		IF rtExecute.Q 
		THEN
			Busy 											:= TRUE;
			Done											:= FALSE;
			Error											:= FALSE;
			ErrorID											:= 0;
			Errortext										:= '';
			CurrState										:= 0;
			linkState										:= 0;
			ReqStateOK										:= FALSE;
			MEMSET(ADR(StateBits),0,SIZEOF(StateBits));
			MEMSET(ADR(CrcError),0,SIZEOF(CrcError));	
			StateText										:= '';
	
			SetSlaveSTATE(bExecute := FALSE, sNetId:= EcMasterAmsNetId,nSlaveAddr:= SlaveAddr);
			GetSlaveSTATE(bExecute := FALSE,sNetId:= EcMasterAmsNetId,nSlaveAddr:= SlaveAddr);
			GetSlaveCrcErrorEx(bExecute := FALSE,sNetId:= EcMasterAmsNetId,nSlaveAddr:= SlaveAddr);

			IF(ReqState <> CurrState
				OR ReqState <> MemReqState)
				AND ReqState <> 0
			THEN
				SetSlaveState(bExecute:= TRUE,reqState:= ReqState);
				MemReqState 								:= ReqState;
				state 										:= 10;

			ELSE
				(* Start Reading State *)
				GetSlaveState(bExecute	:= TRUE);
				state 										:= 1;
			END_IF

		ELSIF NOT Execute 
		THEN
			Done 											:= FALSE;
			Error											:= FALSE;
			ErrorID											:= 0;
			ErrorText										:= '';
		END_IF

	(* Read Slave State **************************************)
	1:
		(* Work block *)
		GetSlaveState();

		IF NOT GetSlaveState.bBusy
		THEN
			IF GetSlaveState.bError THEN
				Busy										:= FALSE;
				Error										:= TRUE;
				ErrorId										:= GetSlaveState.nErrId;
				ErrorText									:= CONCAT('FB_EcGetSlaveSTATE Id: ',UDINT_TO_STRING(ErrorId));
				state 										:= 0;
			ELSE       
				ReqStateOK 									:= (ReqState = CurrState OR ReqState = 0);         					
				CurrState 									:= GetSlaveState.state.deviceState;
				linkState 									:= GetSlaveState.State.linkState;
				StateText 									:= F_ConvStateToString(GetSlaveState.State.deviceState);
			 	StateBits							 		:= F_ConvSlaveStateToBitsEx(GetSlaveState.state);
				state										:= state + 1;
			END_IF
			GetSlaveSTATE(bExecute := FALSE);
		ELSE
			;
		END_IF

	(* Read Slave CRC Error Counter  **************************************)		
	2: 
		(* Work block *)
		GetSlaveCrcErrorEx();

		IF NOT GetSlaveCrcErrorEx.bBusy
		THEN
			IF GetSlaveCrcErrorEx.bError THEN
				Busy										:= FALSE;
				Error										:= TRUE;
				ErrorId										:= GetSlaveCrcErrorEx.nErrId;
				ErrorText									:= CONCAT('FB_EcGetSlaveCrcErrorEx Id: ',UDINT_TO_STRING(ErrorId));
				state 										:= 0;
			ELSE       
				CrcError									:= 	GetSlaveCrcErrorEx.crcError;
				Done 										:= TRUE;
				Busy 										:= FALSE;
				state										:= 0;
			END_IF
			GetSlaveCrcErrorEx(bExecute := FALSE);
		ELSE
			;
		END_IF

	(* Set state  *****************************************)
	10:	
		SetSlaveState();  
		IF NOT SetSlaveState.bBusy
		THEN
			IF SetSlaveState.bError 
			THEN             	
				Busy										:= FALSE;
				Error										:= TRUE;
				ErrorId										:= SetSlaveState.nErrId;
				ErrorText									:= CONCAT('FB_EcSetSlaveSTATE Id: ',UDINT_TO_STRING(ErrorId));
				state 										:= 0;
			ELSIF SetSlaveState.CurrState.deviceState = MemReqState 
			THEN
				ReqStateOK									:= TRUE;
				Busy 										:= FALSE;
				Done 										:= TRUE;	
				state 										:= 0;
			ELSE                    				
				Busy										:= FALSE;		
				Error										:= TRUE;
				ErrorId										:= E_AdsErr.DEVICE_ABORTED;
				ErrorText									:= 'SetSlaveState DEVICESTATE <> ReqState';
				state	 									:= 0;
			END_IF         					
			CurrState 										:= SetSlaveState.currState.deviceState;
			linkState 										:= SetSlaveState.currState.linkState;
			StateText 										:= F_ConvStateToString(SetSlaveState.currState.deviceState);
			StateBits							 			:= F_ConvSlaveStateToBitsEx(SetSlaveState.currState);
			SetSlaveState(bExecute := FALSE);              						
		END_IF                      						
	END_CASE


(*********************************************************************)

END_FUNCTION_BLOCK

// ---- POUs/FileHandling/Basic/FileHandling.TcPOU
{attribute 'no_check'}
//Wrapper for all file fucntions provided by lib Tc2_TcSystem.Lib, see Beckhoff information system for detailed information of each function. 
FUNCTION_BLOCK FileHandling EXTENDS FbBase
VAR_OUTPUT CONSTANT
	FNC_OPEN												:	INT := 0; //With this function a new file can be created, or a closed existing file can be re-opened for further processing
	FNC_READ												:	INT := 1; //With this function  the contents of an already opened file can be read. The file must have been already opened for read access
	FNC_WRITE												:	INT := 2; //Data can be written into a file with this function if it is opened in write mode
	FNC_PUTS												:	INT := 3; //The function writes strings to the file if it is opened in write mode
	FNC_GETS												:	INT := 4; //The function reads zero terminated strings from a file and moves the file pointer to the next line.(if pBuffer is <> 0, the read line will copied to the buffer as well)
	FNC_CLOSE												:	INT := 5; //With this function the file can be closed, and thereby placed into a defined state for further processing by other programs
	FNC_DELETE												:	INT := 6; //With this function the existing file can be deleted
	FNC_RENAME												:	INT := 7; //With this function the existing file can be renamed.
	FNC_REMOVEDIR											:	INT := 8; //This function removes a directory from the data medium. A directory containing data can not be removed!
	FNC_CREATEDIR											:	INT := 9; //This function creates new directories on the data medium.
	FNC_SEEK												:	INT := 10;//With this function the file pointer of an opened file can be set to a definable position
	FNC_TELL												:	INT := 11;//The function gets the current position of the file pointer. The position is expressed as an offset relative to the beginning of the stream.
	FNC_EOF													:	INT := 12;//The function tests for the end-of-file.
	FNC_LOAD												:	INT := 13;//The file is opened implicitly in binary mode, the contents are read out and the file is then closed again.
END_VAR             										                 										
VAR_INPUT           										
	Fnc														:	INT (FNC_OPEN..FNC_LOAD) := FNC_OPEN; //Parameter for requested function
	AMSNetId												:	T_AmsNetId := ''; //Ams Net Id 
	Timeout													:	TIME := DEFAULT_ADS_TIMEOUT; //Ads timeout 
	Mode													:	DWORD := FOPEN_MODEAPPEND OR FOPEN_MODEPLUS OR FOPEN_MODETEXT; 
																			(* 	FOPEN_MODEREAD "r": Opens for reading. If the file does not exist or cannot be found, the call fails.
																				FOPEN_MODEWRITE  "w": Opens an empty file for writing. If the given file exists, its contents are destroyed.
																				FOPEN_MODEAPPEND  "a": Opens for writing at the end of the file (appending) without removing the EOF marker before writing new data to the file; creates the file first if it doesn’t exist.
																				FOPEN_MODEREAD OR FOPEN_MODEPLUS  "r+": Opens for reading and writing. The file must exist.
																				FOPEN_MODEWRITE OR FOPEN_MODEPLUS  "w+": Opens an empty file for both reading and writing. If the given file exists, its contents are destroyed.
																				FOPEN_MODEAPPEND OR FOPEN_MODEPLUS  "a+": 	Opens for reading and appending; the appending operation includes the removal of the EOF marker before new data is written to the file and the EOF marker is restored after writing is complete; creates the file first if it doesn’t exist.
																															When a file is opened with the "a" or "a+" access type, all write operations occur at the end of the file. The file pointer can be repositioned using FB_FileSeek, but is always moved back to the end of the file before any write operation is carried out. Thus, existing data cannot be overwritten. 																				                                    								
																				FOPEN_MODEBINARY  "b": Open in binary (untranslated) mode.
																				FOPEN_MODETEXT  "t": Open in text (translated) mode. *)
	Path													:	T_MaxString; // \\PC-Name\Folder\ 
	FileName												:	T_MaxString := ''; // NewFile.xyz 
	OldFileName												:	T_MaxString := ''; // File.xyz 
	pBuffer													:	PVOID; //pointer to data section 
	Length													: 	UDINT; // sizeof data section for read and write. Note to use "LEN" while writing-command, beacause otherwise the whole datasection and not only the string will be written 
	SeekOrigin												: 	E_SeekOrigin := SEEK_SET; //Seek function parameter - Contains the relative position for the move.
	SeekPos													:	DINT; //Seek function parameter - Contains the desired (new) target position of the file pointer.
END_VAR
VAR_OUTPUT
	EOF														:	BOOL;	//This output is switched to TRUE if the end of file is reached.
	WorkedLen												:	UDINT;	//Contains the number of bytes currently read or written
	hFile													:	UINT;	//File handle of currently opened file
	ActSeekPos												:	DINT;	//Act file pointer position of filled by Tell function
	Line   													: T_MaxString; //Read line of file - filled by function Gets

END_VAR
VAR
(* internal used variables ************************************************************)
	MemErrorText											:	STRING(50);
	MemFnc													:	INT := -1;
	
(* trigger ******************************************************************************)

(* function-block instances ************************************************************)
	File_Open												:	FB_FileOpen;
	File_Close												: 	FB_FileClose;
	File_Read 												: 	FB_FileRead;
	File_Write												:	FB_FileWrite;
	File_Delete												:	FB_FileDelete;
	File_Rename												:	FB_FileRename;
	File_Puts												:	FB_FilePuts;
	File_Gets												:	FB_FileGets;
	File_CreateDir											:	FB_CreateDir;
	File_RemoveDir											:	FB_RemoveDir;
	File_Tell												:	FB_FileTell ;
	File_Seek												:	FB_FileSeek ;
	File_EoF												:	FB_EOF;
	File_Load												:	FB_FileLoad;
END_VAR

	(* FileHandling												V2.0	*)
	(********************************************************************)

(* Sequence **********************************************************************)
	rtExecute(CLK := Execute);
	IF rtExecute.Q
		AND MemFnc < 0
	THEN
		Busy												:= TRUE;
		Done												:= FALSE;
		Error												:= FALSE;
		ErrorId												:= 0;
		CASE fnc OF                     					
		FNC_OPEN:		MemFnc 								:= fnc;
		FNC_READ:		MemFnc 								:= fnc;
		FNC_WRITE:		MemFnc 								:= fnc;
		FNC_PUTS:		MemFnc 								:= fnc;
		FNC_GETS:		MemFnc 								:= fnc;
		FNC_CLOSE:		MemFnc 								:= fnc;
		FNC_DELETE:		MemFnc 								:= fnc;
		FNC_RENAME:		MemFnc 								:= fnc;
		FNC_REMOVEDIR: 	MemFnc 								:= fnc;
		FNC_CREATEDIR: 	MemFnc 								:= fnc;
		FNC_SEEK:		MemFnc 								:= fnc;
		FNC_TELL:		MemFnc 								:= fnc;
		FNC_EOF:		MemFnc 								:= fnc;
		FNC_LOAD:		MemFnc 								:= fnc;
		ELSE                            					
			ErrorId											:= E_AdsErr.DEVICE_INVALIDPARM;
			Error											:= TRUE;
			Done											:= FALSE;
			Busy											:= FALSE;
		END_CASE
	END_IF

	CASE MemFnc OF
		FNC_OPEN:		Open(Execute := Execute);
		FNC_READ:		Read(Execute := Execute);
		FNC_WRITE:		Write(Execute := Execute);
		FNC_PUTS:		Puts(Execute := Execute);
		FNC_GETS:		Gets(Execute := Execute);
		FNC_CLOSE:		Close(Execute := Execute);
		FNC_DELETE:		Delete(Execute := Execute);
		FNC_RENAME:		Rename(Execute := Execute);
		FNC_REMOVEDIR: 	RemoveDir(Execute := Execute);
		FNC_CREATEDIR: 	CreateDir(Execute := Execute);
		FNC_SEEK:		Seek(Execute := Execute);
		FNC_TELL:		Tell(Execute := Execute);
		FNC_EOF:		IsEof(Execute := Execute);
		FNC_LOAD:		Load(Execute := Execute);
	
	-1:
		IF NOT Execute
		THEN
			Busy											:= FALSE;
			Done											:= FALSE;
			Error											:= FALSE;
			ErrorID											:= 0;
		END_IF
	END_CASE
(*************************************************************************)

METHOD PUBLIC close : Bool //Return value = TRUE if busy
VAR_INPUT
	Execute		:	BOOL	:= FALSE;
END_VAR
	IF Execute
	THEN
		Error												:=	FALSE;
		ErrorId												:= 0;
		File_Close.bExecute 								:= TRUE;
	ELSIF NOT File_Close.bBusy      						
	THEN                            						
		Error												:=	FALSE;
		ErrorId												:= 0;
		File_Close.bExecute 								:= FALSE;
	END_IF                          						
                                    	
	MemFnc 													:= FNC_CLOSE;
	THIS^.Execute											:= Execute;

	File_Close(
		sNetId		:= AMSNetId,
		hFile		:= hFile,
		bExecute	:= ,
		tTimeout	:= Timeout,
		bBusy		=> Busy,
		bError		=> ,
		nErrId		=> );

	IF NOT File_Close.bBusy
		AND NOT File_Close.bError
		AND File_Close.bExecute
	THEN
		Done												:= TRUE;
		hFile 												:= 0;
	ELSE                            						
		Done												:= FALSE;
	END_IF

	IF NOT Busy
	THEN
		IF File_Close.bExecute
		THEN
			Error											:=	File_Close.bError;
			ErrorId											:= File_Close.nErrId;
		END_IF
		IF NOT Execute
		THEN
			MemFnc											:=  -1;
			File_Close(bExecute 							:= FALSE);
		END_IF
	END_IF

	(* Fehler speichern *)
	IF Error
	THEN
		MemErrorText										:= CONCAT('File_Close ErrorID: ', UDINT_TO_STRING(ErrorID));
	END_IF
	
	Close													:= Busy;
END_METHOD

METHOD PUBLIC createDir : BOOL //Return value = TRUE if busy
//required parameter
//Path
VAR_INPUT
	Execute													:	BOOL;
END_VAR
	IF Execute
	THEN
		Error												:=	FALSE;
		ErrorId												:= 0;
		File_CreateDir.bExecute 							:= TRUE;
	ELSIF NOT File_CreateDir.bBusy      					
	THEN                                					
		Error												:=	FALSE;
		ErrorId												:= 0;
		File_CreateDir.bExecute								:= FALSE;
	END_IF                              					
                                        	
	MemFnc 													:= FNC_CREATEDIR;
	THIS^.Execute											:= Execute;

	File_CreateDir(
		sNetId		:= AMSNetId,
		sPathName	:= Path,
		ePath		:= ,
		bExecute	:= ,
		tTimeout	:= Timeout,
		bBusy		=> Busy,
		bError		=> ,
		nErrId		=> );

	Done													:= NOT File_CreateDir.bBusy
																AND NOT File_CreateDir.bError
																AND File_CreateDir.bExecute;
	IF NOT Busy
	THEN
		IF File_CreateDir.bExecute
		THEN
			Error											:=	File_CreateDir.bError;
			ErrorId											:= File_CreateDir.nErrId;
		END_IF
		IF NOT Execute
		THEN
			MemFnc											:=  -1;
			File_CreateDir(bExecute := FALSE);
		END_IF
	END_IF


	IF Error
	THEN
		MemErrorText										:= CONCAT('File_CreateDir ErrorID: ', UDINT_TO_STRING(ErrorID));
	END_IF
	
	CreateDir												:= Busy;
END_METHOD

METHOD PUBLIC delete : BOOL //Return value = TRUE if busy
//required parameter
//Path
//FileName
VAR_INPUT
	Execute			:	bool;
END_VAR
	IF Execute
	THEN
		Error												:=	FALSE;
		ErrorId												:= 0;
		File_Delete.bExecute 								:= TRUE;
	ELSIF NOT File_Delete.bBusy         					
	THEN                                					
		Error												:=	FALSE;
		ErrorId												:= 0;
		File_Delete.bExecute 								:= FALSE;
	END_IF                              					
                                        	
	MemFnc 													:= FNC_DELETE;
	THIS^.Execute											:= Execute;

	File_Delete(
		sNetId		:= AMSNetId,
		sPathName	:= CONCAT(Path,FileName),
		ePath		:= ,
		bExecute	:= ,
		tTimeout	:= Timeout,
		bBusy		=> Busy,
		bError		=> ,
		nErrId		=> );

	Done													:= 	NOT File_Delete.bBusy
																AND NOT File_Delete.bError
																AND File_Delete.bExecute;
	IF NOT Busy
	THEN
		IF File_Delete.bExecute
		THEN
			Error											:=	File_Delete.bError;
			ErrorId											:= File_Delete.nErrId;
		END_IF
		IF NOT Execute
		THEN
			MemFnc											:= -1;
			File_Delete(bExecute := FALSE);
		END_IF
	END_IF


	IF Error
	THEN
		MemErrorText										:= CONCAT('File_Delete ErrorID: ', UDINT_TO_STRING(ErrorID));
	End_if
	
	Delete													:= Busy;
END_METHOD

METHOD PUBLIC gets : BOOL //Return value = TRUE if busy
//required parameter
//Path
//Filename
//Mode
//pBuffer
VAR_INPUT
	Execute			:	BOOL;
END_VAR
IF pBuffer = 0 THEN
	Busy													:= NOT Error;
	Error													:= TRUE;
	ErrorId													:= E_AdsErr.DEVICE_INVALIDPARM;
	Done													:= FALSE;
	MemFnc													:= -1 ;
	RETURN;                             					
END_IF                                  					
                                        					
	MemFnc 													:= FNC_GETS;
	THIS^.Execute											:= Execute;
                                        					
	CASE State OF                       	
	0:                                  	
		IF Execute                      	
		THEN                            	
			Done											:= FALSE;
			Error											:= FALSE;
			ErrorId 										:= 0;
			
			File_Open(bExecute := FALSE);
			File_Gets(bExecute := FALSE);
			File_Close(bExecute := FALSE);
			
			EOF												:= FALSE;
			WorkedLen										:= 0;
			
			IF hFile = 0
			THEN
				File_Open(
					sNetId		:= AMSNetId,
					sPathName	:= CONCAT(Path,FileName),
					nMode		:= Mode ,
					ePath		:= (* Default *),
					bExecute	:= TRUE,
					tTimeout	:= Timeout,
					bBusy		=> ,
					bError		=> ,
					nErrId		=> ,
					hFile		=> );

				State 										:= 10;
			ELSE                							
				State 										:= 10;
			END_IF
		ELSE
			Done											:= FALSE;
			Error											:= FALSE;
			ErrorId 										:= 0;
		END_IF

	10:
		File_Open();

		IF NOT File_Open.bBusy
		THEN
			IF File_Open.bError
			THEN
				State 										:= 99;
			ELSE
				IF File_Open.bExecute THEN hFile := File_Open.hFile; END_IF
				File_Gets(
					sNetId		:= AMSNetId,
					hFile		:= hFile,
					bExecute	:= TRUE,
					tTimeout	:= Timeout,
					sLine		=> ,
					bEOF		=> ,
					bBusy		=> ,
					bError		=> ,
					nErrId		=> );

				State 										:= 20;
			END_IF
		END_IF

	20:
		File_Gets(bEOF		=> EOF);
		IF NOT File_Gets.bBusy
		THEN
			IF NOT File_Gets.bError
			THEN
				IF pBuffer <> 0 AND Length <> 0
				THEN
					 MEMCPY(pBuffer , ADR(File_Gets.sLine), MIN(TO_UDINT(Length), SIZEOF(File_Gets.sLine)));
				END_IF
				Line										:= File_Gets.sLine;
			END_IF
			IF File_Open.bExecute
			THEN
				File_Close(
					sNetId	:= AMSNetId,
					hFile	:= hFile,
					bExecute:= TRUE,
					tTimeout:= Timeout,
					bBusy	=> ,
					bError	=> ,
					nErrId	=> );
				State										:= 30;
			ELSE
				State										:= 99;
			END_IF

		END_IF

	30:
		File_Close();
		IF NOT File_Close.bBusy
		THEN
			hFile											:= 0;
			State											:= 99;
		END_IF

	99:
		IF NOT Execute
		THEN
			Memfnc											:= -1;
			state 											:= 0;
		END_IF
	END_CASE

	Done													:= state = 99
																AND NOT File_Gets.bError
																AND NOT File_Close.bError
																AND NOT File_Open.bError;
                                        					
	Error													:= state = 99
																AND(
																File_Gets.bError
																OR File_Close.bError
																OR File_Open.bError);
                                        					
	Busy													:= state <> 0
																AND NOT Done
																AND NOT Error;

	IF Error
	THEN
		IF File_Close.bError 	THEN 	ErrorId :=  File_Close.nErrId; 	END_IF
		IF File_Gets.bError 	THEN 	ErrorId :=  File_Gets.nErrId; 	END_IF
		IF File_Open.bError 	THEN	ErrorId :=  File_Open.nErrId; 	END_IF
	ELSE
		ErrorId 											:= 0;
	END_IF                              					
                                        					
	IF NOT Execute                      					
		AND state = 99                  					
	THEN                                					
			MemFnc											:= -1;
		state 												:= 0;
	END_IF                              	
                                        	
	IF Error                            	
	THEN                                	
		MemErrorText										:= CONCAT('File_Gets ErrorID: ', UDINT_TO_STRING(ErrorID));
	END_IF                              					
                                        					
	Gets													:= Busy;
END_METHOD

METHOD PUBLIC isEoF : BOOL //Return value = TRUE if busy
VAR_INPUT
	Execute													:	BOOL;
END_VAR
	IF Execute
	THEN
		Error												:=	FALSE;
		ErrorId												:= 0;
		File_EoF.bExecute 									:= TRUE;
	ELSIF NOT File_EoF.bBusy           					
	THEN                                					
		Error												:=	FALSE;
		ErrorId												:= 0;
		File_EoF.bExecute 									:= FALSE;
	END_IF                              							
	                                    	
	MemFnc 													:= FNC_EOF;
	THIS^.Execute											:= Execute;
                                        	
	File_EoF(
		sNetId		:= AMSNetId,
		hFile		:= hFile ,
		tTimeout	:= Timeout,
		bBusy		=> Busy,
		bError		=> ,
		nErrId		=> ,
		bEoF		=> EoF);

	Done													:= NOT File_EoF.bBusy
																AND NOT File_EoF.bError
																AND File_EoF.bExecute;
	IF NOT Busy                         					
	THEN                        					
		IF File_EoF.bExecute           					
		THEN                            	
			Error											:=	File_EoF.bError;
			ErrorId											:= File_EoF.nErrId;
		END_IF
		IF NOT Execute
		THEN
			MemFnc											:= 1;
			File_EoF(bExecute := FALSE);
		END_IF
	END_IF


	IF Error
	THEN
		MemErrorText										:= CONCAT('File_EoF ErrorID: ', UDINT_TO_STRING(ErrorID));
	END_IF
	
	IsEoF													:= Busy;
END_METHOD

METHOD PUBLIC load : BOOL //Result = Busy
//required parameter
//Path
//FileName
VAR_INPUT
	Execute				:	BOOL; 
END_VAR
IF Execute
THEN
	Error													:= FALSE;
	ErrorId													:= 0;
	File_Load.bExecute 										:= TRUE;
ELSIF NOT File_Load.bBusy           						
THEN                                						
	Error													:=	FALSE;
	ErrorId													:= 0;
	File_Load.bExecute 										:= FALSE;
END_IF	

MemFnc 														:= FNC_LOAD;
THIS^.Execute												:= Execute;

(* Work File Load *)
File_Load(
	sNetId		:= AMSNetId, 
	sPathName	:= CONCAT(Path,FileName), 
	pReadBuff	:= pBuffer, 
	cbReadLen	:= Length, 
	bExecute	:= , 
	tTimeout	:= Timeout, 
	bBusy		=> Busy, 
	bError		=> , 
	nErrId		=> , 
	cbRead		=> WorkedLen);
Done														:= NOT File_Load.bBusy
																AND NOT File_Load.bError
																AND File_Load.bExecute;
IF NOT Busy
THEN
	IF File_Load.bExecute
	THEN
		Error												:= File_Load.bError;
		ErrorId												:= File_Load.nErrId;
	END_IF
	IF NOT Execute
	THEN
		MemFnc												:= -1;
		File_Load(bExecute := FALSE);
	END_IF
END_IF

IF Error
THEN
	MemErrorText											:= CONCAT('File_Load ErrorID: ', UDINT_TO_STRING(ErrorID));
END_IF                              						
                                    	
load														:= Busy;
END_METHOD

METHOD PUBLIC open : BOOL //Return value = TRUE if busy
//required parameter
//Path
//FileName
//Mode
VAR_INPUT
	Execute				:	BOOL; 
END_VAR
IF Execute
THEN
	Error													:= FALSE;
	ErrorId													:= 0;
	File_Open.bExecute 										:= TRUE;
ELSIF NOT File_Open.bBusy           						
THEN                                						
	Error													:=	FALSE;
	ErrorId													:= 0;
	File_Open.bExecute 										:= FALSE;
END_IF	

MemFnc 														:= FNC_OPEN;
THIS^.Execute												:= Execute;

(* Work File Open *)
File_Open(
	sNetId		:= AMSNetId,
	sPathName	:= CONCAT(Path,FileName),
	nMode		:= Mode ,
	ePath		:= (* Default *),
	bExecute	:= ,
	tTimeout	:= Timeout,
	bBusy		=> Busy,
	bError		=> ,
	nErrId		=> ,
	hFile		=> hFile);

Done														:= NOT File_Open.bBusy
																AND NOT File_Open.bError
																AND File_Open.bExecute;
IF NOT Busy
THEN
	IF File_Open.bExecute
	THEN
		Error												:=	File_Open.bError;
		ErrorId												:= File_Open.nErrId;
	END_IF
	IF NOT Execute
	THEN
		MemFnc												:= -1;
		File_Open(bExecute := FALSE);
	END_IF
END_IF

IF Error
THEN
	MemErrorText											:= CONCAT('File_Open ErrorID: ', UDINT_TO_STRING(ErrorID));
END_IF                              						
                                    	
Open														:= Busy;
END_METHOD

METHOD PUBLIC puts : BOOL //Return value = TRUE if busy
//required parameter
//Path
//FileName
//Mode
//pBuffer
//Lenght
VAR_INPUT
	Execute				:	BOOL;
END_VAR
IF pBuffer = 0 THEN
	Busy													:= NOT Error;
	Error													:= TRUE;
	ErrorId													:= E_AdsErr.DEVICE_INVALIDPARM;
	Done													:= FALSE;
	MemFnc													:= -1 ;
	RETURN;
END_IF

	MemFnc 													:= FNC_PUTS;
	THIS^.Execute											:= Execute;

	CASE State OF
	0:
		IF Execute
		THEN
			Done											:= FALSE;
			Error											:= FALSE;
			ErrorId 										:= 0;
			
			File_Open(bExecute := FALSE);
			File_Puts(bExecute := FALSE);
			File_Close(bExecute := FALSE);
			
			EOF												:= FALSE;
			WorkedLen										:= 0;
			
			IF hFile = 0
			THEN
				File_Open(
					sNetId		:= AMSNetId,
					sPathName	:= CONCAT(Path,FileName),
					nMode		:= Mode ,
					ePath		:= (* Default *),
					bExecute	:= TRUE,
					tTimeout	:= Timeout,
					bBusy		=> ,
					bError		=> ,
					nErrId		=> ,
					hFile		=> );

				State 										:= 10;
			ELSE                							
				State 										:= 10;
			END_IF              							
		ELSE                    							
			Done											:= FALSE;
			Error											:= FALSE;
			ErrorId 										:= 0;
		END_IF

	10:
		File_Open();

		IF NOT File_Open.bBusy
		THEN
			IF File_Open.bError
			THEN
				State 										:= 99;
			ELSE
				IF File_Open.bExecute THEN hFile := File_Open.hFile; END_IF
				MEMCPY(ADR(File_Puts.sLine),  pBuffer, MIN(TO_UDINT(Length), SIZEOF(File_Puts.sLine)));
				File_Puts(
					sNetId		:= AMSNetId,
					hFile		:= hFile,
					sLine		:= (* siehe oben *),
					bExecute	:= TRUE,
					tTimeout	:= Timeout,
					bBusy		=> ,
					bError		=> ,
					nErrId		=> );

				State 										:= 20;
			END_IF
		END_IF

	20:
		MEMCPY(ADR(File_Puts.sLine),  pBuffer, MIN(TO_UDINT(Length), SIZEOF(File_Puts.sLine)));
		File_Puts();

		IF NOT File_Puts.bBusy
		THEN
			IF File_Open.bExecute
			THEN
				File_Close(
					sNetId	:= AMSNetId,
					hFile	:= hFile,
					bExecute:= TRUE,
					tTimeout:= Timeout,
					bBusy	=> ,
					bError	=> ,
					nErrId	=> );
				State										:= 30;
			ELSE
				State										:= 99;
			END_IF

		END_IF

	30:
		File_Close();
		IF NOT File_Close.bBusy
		THEN
			hFile						:= 0;
			State						:= 99;
		END_IF

	99:
		IF NOT Execute
		THEN
			Memfnc					:= -1;
			state 					:= 0;
		END_IF
	END_CASE

	Done							:= state = 99
										AND NOT File_Puts.bError
										AND NOT File_Close.bError
										AND NOT File_Open.bError;

	Error							:= state = 99
										AND(
										File_Puts.bError
										OR File_Close.bError
										OR File_Open.bError);

	Busy							:= state <> 0
										AND NOT Done
										AND NOT Error;

	IF Error
	THEN
		IF File_Close.bError 	THEN	ErrorId :=  File_Close.nErrId; 	END_IF
		IF File_Puts.bError 	THEN 	ErrorId :=  File_Puts.nErrId; 	END_IF
		IF File_Open.bError 	THEN 	ErrorId :=  File_Open.nErrId;	END_IF
	ELSE
		ErrorId 					:= 0;
	END_IF

	IF NOT Execute
		AND state = 99
	THEN
		MemFnc						:= -1;
		state 						:= 0;
	END_IF

	IF Error
	THEN
		MemErrorText				:= CONCAT('File_Puts ErrorID: ', UDINT_TO_STRING(ErrorID));
	END_IF
	
	Puts							:= Busy;
END_METHOD

METHOD PUBLIC read : BOOL //Return value = TRUE if busy
//required parameter
//Path
//FileName
//Mode
//pBuffer
//Lenght
VAR_INPUT
	Execute			:	BOOL;
END_VAR
IF pBuffer = 0 THEN
	Busy													:= NOT Error;
	Error													:= TRUE;
	ErrorId													:= E_AdsErr.DEVICE_INVALIDPARM;
	Done													:= FALSE;
	MemFnc													:= -1 ;
	RETURN;                             					
END_IF                                  					
                                        	
	MemFnc 													:= FNC_READ;
	THIS^.Execute											:= Execute;

	CASE State OF
	0:
		IF Execute
		THEN
			Done											:= FALSE;
			Error											:= FALSE;
			ErrorId 										:= 0;
			
			File_Open(bExecute := FALSE);
			File_Read(bExecute := FALSE);
			File_Close(bExecute := FALSE);
			
			EOF												:= FALSE;
			WorkedLen										:= 0;
			
			IF hFile = 0
			THEN
				File_Open(
					sNetId		:= AMSNetId,
					sPathName	:= CONCAT(Path,FileName),
					nMode		:= Mode ,
					ePath		:= (* Default *),
					bExecute	:= TRUE,
					tTimeout	:= Timeout,
					bBusy		=> ,
					bError		=> ,
					nErrId		=> ,
					hFile		=> );

				State 										:= 10;
			ELSE                    						
				State 										:= 10;
			END_IF                  						
		ELSE                        						
			Done											:= FALSE;
			Error											:= FALSE;
			ErrorId 										:= 0;
		END_IF

	10:
		File_Open();
		IF NOT File_Open.bBusy
		THEN
			IF File_Open.bError
			THEN
				State 										:= 99;
			ELSE
				IF File_Open.bExecute THEN hFile := File_Open.hFile; END_IF
				File_Read(
					sNetId		:= AmsNetId,
					hFile		:= hFile,
					pReadBuff	:= pBuffer,
					cbReadLen	:= Length,
					bExecute	:= TRUE,
					tTimeout	:= Timeout,
					bBusy		=> ,
					bError		=> ,
					nErrId		=> ,
					cbRead		=> ,
					bEOF		=> );

				State 										:= 20;
			END_IF
		END_IF

	20:
		File_Read(
			pReadBuff	:= pBuffer,
			cbReadLen	:= Length,
			bExecute	:= TRUE,
			cbRead		=> WorkedLen,
			bEOF		=> EOF);

		IF NOT File_Read.bBusy
		THEN
			IF File_Open.bExecute
			THEN
				File_Close(
					sNetId	:= AMSNetId,
					hFile	:= hFile,
					bExecute:= TRUE,
					tTimeout:= Timeout,
					bBusy	=> ,
					bError	=> ,
					nErrId	=> );
				State										:= 30;
			ELSE                        						
				State										:= 99;
			END_IF                      						
                                        						
		END_IF                          						
                                        						
	30:                                 						
		File_Close();                   						
		IF NOT File_Close.bBusy         						
		THEN                            						
			hFile											:= 0;
			State											:= 99;
		END_IF                          						
                                        						
	99:                                 						
		IF NOT Execute                  						
		THEN                            				
			Memfnc											:= -1;
			state 											:= 0;
		END_IF                          	
	END_CASE                            	
                                        	
	Done													:= state = 99
																AND NOT File_Read.bError
																AND NOT File_Close.bError
																AND NOT File_Open.bError;
	                                    						
	Error													:= state = 99
																AND(
																File_Read.bError
																OR File_Close.bError
																OR File_Open.bError);
	                                    						
	Busy													:= state <> 0
																AND NOT Done
																AND NOT Error;

	IF Error
	THEN
		IF File_Close.bError	THEN 	ErrorId :=  File_Close.nErrId;	END_IF
		IF File_Read.bError 	THEN	ErrorId :=  File_Read.nErrId; 	END_IF
		IF File_Open.bError		THEN	ErrorId :=  File_Open.nErrId; 	END_IF
	ELSE
		ErrorId 											:= 0;
	END_IF                              						
                                        						
	IF NOT Execute                      						
		AND state = 99                  						
	THEN                                						
		MemFnc												:=  -1;
		state 												:= 0;
	END_IF                              	
                                        	
	IF Error                            	
	THEN                                	
		MemErrorText										:= CONCAT('File_Read ErrorID: ', UDINT_TO_STRING(ErrorID));
	END_IF                              						
	                                    						
	Read													:= Busy;
END_METHOD

METHOD PUBLIC removeDir : BOOL //Return value = TRUE if busy
//required parameter
//Path
VAR_INPUT
	Execute				:	BOOL;
END_VAR
	IF Execute
	THEN
		Error												:= FALSE;
		ErrorId												:= 0;
		File_RemoveDir.bExecute 							:= TRUE;
	ELSIF NOT File_RemoveDir.bBusy      					
	THEN                                					
		Error												:=	FALSE;
		ErrorId												:= 0;
		File_RemoveDir.bExecute 							:= FALSE;
	END_IF                              					
                                        	
	MemFnc 													:= FNC_REMOVEDIR;
	THIS^.Execute											:= Execute;

	File_RemoveDir(
		sNetId		:= AMSNetId,
		sPathName	:= Path,
		ePath		:= ,
		bExecute	:= ,
		tTimeout	:= Timeout,
		bBusy		=> Busy,
		bError		=> ,
		nErrId		=> );

	Done													:= NOT File_RemoveDir.bBusy
																AND NOT File_RemoveDir.bError
																AND File_RemoveDir.bExecute;
	IF NOT Busy                         					
	THEN                                					
		IF File_RemoveDir.bExecute      					
		THEN                            					
			Error											:=	File_RemoveDir.bError;
			ErrorId											:= File_RemoveDir.nErrId;
		END_IF                          	
		IF NOT Execute                  	
		THEN                            	
			MemFnc											:=  -1;
			File_RemoveDir(bExecute := FALSE);
		END_IF
	END_IF


	IF Error
	THEN
		MemErrorText										:= CONCAT('File_RemoveDir ErrorID: ', UDINT_TO_STRING(ErrorID));
	END_IF                              					
	                                    	
	RemoveDir												:= Busy;
END_METHOD

METHOD PUBLIC rename : BOOL //Return value = TRUE if busy
//required parameter
//Path
//OldFileName
//FileName
VAR_INPUT
	Execute			:	BOOL;
END_VAR
	IF Execute
	THEN
		Error												:=	FALSE;
		ErrorId												:= 0;
		File_Rename.bExecute 								:= TRUE;
	ELSIF NOT File_Rename.bBusy         					
	THEN                                					
		Error												:=	FALSE;
		ErrorId												:= 0;
		File_Rename.bExecute 								:= FALSE;
	END_IF                              					
                                        	
	MemFnc 													:= FNC_RENAME;
	THIS^.Execute											:= Execute;

	File_Rename(
		sNetId		:= AMSNetId,
		sOldName	:= CONCAT(Path,OldFileName),
		sNewName	:= CONCAT(Path,FileName),
		ePath		:= ,
		bExecute	:=	,
		tTimeout	:=	Timeout,
		bBusy		=> Busy,
		bError		=> ,
		nErrId		=> );

	Done													:= NOT File_Rename.bBusy
																AND NOT File_Rename.bError
																AND File_Rename.bExecute;
	IF NOT Busy                         					
	THEN                                					
		IF File_Rename.bExecute         					
		THEN                            	
			Error											:=	File_Rename.bError;
			ErrorId											:= File_Rename.nErrId;
		END_IF
		IF NOT Execute
		THEN
			MemFnc											:= -1;
			File_Rename(bExecute := FALSE);
		END_IF
	END_IF


	IF Error
	THEN
		MemErrorText										:= CONCAT('File_Rename ErrorID: ', UDINT_TO_STRING(ErrorID));
	END_IF
	
	Rename													:= Busy;
END_METHOD

METHOD PUBLIC seek : BOOL //Return value = TRUE if busy
//required parameter
//Path
//SeekPos
//SeekOrigin
VAR_INPUT
	Execute			:	BOOL;
END_VAR
	IF Execute
	THEN
		Error												:=	FALSE;
		ErrorId												:= 0;
		File_Seek.bExecute 									:= TRUE;
	ELSIF NOT File_Seek.bBusy           					
	THEN                                					
		Error												:=	FALSE;
		ErrorId												:= 0;
		File_Seek.bExecute 									:= FALSE;
	END_IF                              							
	                                    	
	MemFnc 													:= FNC_SEEK;
	THIS^.Execute											:= Execute;
                                        	
	File_Seek(
		sNetId		:= AMSNetId,
		hFile		:= hFile ,
		nSeekPos	:= SeekPos,
		eOrigin		:= SeekOrigin,
		bExecute	:= ,
		tTimeout	:= Timeout,
		bBusy		=> Busy,
		bError		=> ,
		nErrId		=> );

	Done													:= NOT File_Seek.bBusy
																AND NOT File_Seek.bError
																AND File_Seek.bExecute;
	IF NOT Busy                         					
	THEN                    
		ActSeekPos											:= File_Seek.nSeekPos;           					
		IF File_Seek.bExecute           					
		THEN                            	
			Error											:=	File_Seek.bError;
			ErrorId											:= File_Seek.nErrId;
		END_IF
		IF NOT Execute
		THEN
			MemFnc											:= 1;
			File_Seek(bExecute := FALSE);
		END_IF
	END_IF


	IF Error
	THEN
		MemErrorText										:= CONCAT('File_Seek ErrorID: ', UDINT_TO_STRING(ErrorID));
	END_IF
	
	Seek													:= Busy;
END_METHOD

METHOD PUBLIC tell : BOOL //Return value = TRUE if busy
VAR_INPUT
	Execute													:	BOOL;
END_VAR
	IF Execute
	THEN
		Error												:=	FALSE;
		ErrorId												:= 0;
		File_Tell.bExecute 									:= TRUE;
	ELSIF NOT File_Tell.bBusy           					
	THEN                                					
		Error												:=	FALSE;
		ErrorId												:= 0;
		File_Tell.bExecute 									:= FALSE;
	END_IF                              					
                                        					
	MemFnc 													:= FNC_TELL;
	THIS^.Execute											:= Execute;
                                        			
	File_Tell(                          			
		sNetId		:= AMSNetId,        			
		hFile		:= hFile ,          			
		bExecute	:= ,                			
		tTimeout	:= Timeout,         			
		nSeekPos	=> ActSeekPos,      			
		bBusy		=> Busy,            			
		bError		=> ,                			
		nErrId		=> );               			
                                        			
	Done														:= NOT File_Tell.bBusy
																AND NOT File_Tell.bError
																AND File_Tell.bExecute;
	IF NOT Busy                         						
	THEN                                						
		IF File_Tell.bExecute           						
		THEN                            						
			Error												:=	File_Tell.bError;
			ErrorId												:= File_Tell.nErrId;
		END_IF                          						
		IF NOT Execute                  						
		THEN                            						
			MemFnc												:= -1;
			File_Tell(bExecute := FALSE);               	
		END_IF                                          	
	END_IF                                              	
                                                        	
                                                        	
	IF Error                                            	
	THEN                                                	
		MemErrorText											:= CONCAT('File_Tell ErrorID: ', UDINT_TO_STRING(ErrorID));
	END_IF                                              	
	                                                    	
	Tell 														:= Busy;
END_METHOD

METHOD PUBLIC write : BOOL //Return value = TRUE if busy
//required parameter
//Path
//Filename
//Mode
//pBuffer
//Length
VAR_INPUT
	Execute													:	BOOL;
END_VAR
IF pBuffer = 0 THEN
	Busy													:= NOT Error;
	Error													:= TRUE;
	ErrorId													:= E_AdsErr.DEVICE_INVALIDPARM;
	Done													:= FALSE;
	MemFnc													:= -1 ;
	RETURN;                             					
END_IF                                  					
                                        					
	MemFnc 													:= FNC_WRITE;
	THIS^.Execute											:= Execute;
                                        					
	CASE State OF                       	
	0:                                  	
		IF Execute                      	
		THEN                            	
			Done											:= FALSE;
			Error											:= FALSE;
			ErrorId 										:= 0;
			
			File_Open(bExecute := FALSE);
			File_Write(bExecute := FALSE);
			File_Close(bExecute := FALSE);	
			
			WorkedLen										:= 0;
			
			IF hFile = 0
			THEN
				File_Open(
					sNetId		:= AMSNetId,
					sPathName	:= CONCAT(Path,FileName),
					nMode		:= Mode ,
					ePath		:= (* Default *),
					bExecute	:= TRUE,
					tTimeout	:= Timeout,
					bBusy		=> ,
					bError		=> ,
					nErrId		=> ,
					hFile		=> );

				State 										:= 10;
			ELSE	                    					
				State 										:= 10;
			END_IF                      					
		ELSE                            					
			Done											:= FALSE;
			Error											:= FALSE;
			ErrorId 										:= 0;
		END_IF

	10:
		File_Open(hFile		=> hFile);

		IF NOT File_Open.bBusy
		THEN
			IF File_Open.bError
			THEN
				State 										:= 99;
			ELSE
				IF File_Open.bExecute THEN hFile := File_Open.hFile; END_IF
				File_Write(
					sNetId		:= AMSNetId,
					hFile		:= hFile,
					pWriteBuff	:= pBuffer,
					cbWriteLen	:= Length,
					bExecute	:= TRUE,
					tTimeout	:= Timeout,
					bBusy		=> ,
					bError		=> ,
					nErrId		=> ,
					cbWrite		=> );
				State 										:= 20;
			END_IF
		END_IF

	20:
		File_Write(
			pWriteBuff	:= pBuffer,
			cbWriteLen	:= Length,
			bExecute	:= TRUE,
			cbWrite		=> WorkedLen);

		IF NOT File_Write.bBusy
		THEN
			IF File_Open.bExecute
			THEN
				File_Close(
					sNetId		:= AMSNetId,
					hFile		:= hFile,
					bExecute	:= TRUE,
					tTimeout	:= Timeout,
					bBusy		=> ,
					bError		=> ,
					nErrId		=> );
				State										:= 30;
			ELSE  //Exit without closing the file as the file was opended externaly                     					
				State										:= 99;
			END_IF                  					
		ELSE                            					
			;                           					
		END_IF                          					
                                        	
	30:                                 	
		File_Close();                   	
		IF NOT File_Close.bBusy         	
		THEN                       	
			hFile											:= 0;
			State											:= 99;
		END_IF

	99:
		IF NOT Execute
		THEN	
			Memfnc											:= -1;
			state 											:= 0;
		END_IF
	END_CASE

	Done													:= state = 99
																AND NOT File_Write.bError
																AND NOT File_Close.bError
																AND NOT File_Open.bError;
                                    						
	Error													:= state = 99
																AND(
																File_Write.bError
																OR File_Close.bError
																OR File_Open.bError);
                                    						
	Busy													:= state <> 0
																AND NOT Done
																AND NOT Error;
                                    					
	IF Error
	THEN
		IF File_Close.bError 	THEN 	ErrorId :=  File_Close.nErrId;	END_IF
		IF File_Write.bError 	THEN 	ErrorId :=  File_Write.nErrId;	END_IF
		IF File_Open.bError 	THEN 	ErrorId :=  File_Open.nErrId; 	END_IF
	ELSE
		ErrorId 											:= 0;
	END_IF                          						
                                    						
	IF NOT Execute                  						
		AND state = 99              						
	THEN                            						
		MemFnc												:=  -1;
		state 												:= 0;
	END_IF                          						
                                    	
	IF Error                        	
	THEN                            	
		MemErrorText										:= CONCAT('File_Write ErrorID: ', UDINT_TO_STRING(ErrorID));
	END_IF                          	
	                                	
	Write													:= Busy;
END_METHOD

END_FUNCTION_BLOCK

// ---- POUs/FileHandling/Basic/ReadDirSimpleExt.TcPOU
{attribute 'no_check'}
//List down all files and it's information founded in a directory - specified by file type if needed 
FUNCTION_BLOCK ReadDirSimpleExt EXTENDS FbBase
VAR_OUTPUT CONSTANT
	MIN_ENTRYS												:	INT := 1;	
	MAX_ENTRYS												:	INT := PARAM.READ_DIR_SIMPLE_MAX_ENTRYS;	//see library parameter to customize parameter	
	MAX_STRING_LEN											:	INT := PARAM.READ_DIR_SIMPLE_MAX_STRING_LEN;//see library parameter to customize parameter
END_VAR            										  										
VAR_INPUT           										
	AMSNetId												:	T_AmsNetId; //AMS Net Id
	Timeout													:	TIME := DEFAULT_ADS_TIMEOUT; //ADS Timeout Default 3s 
	Path													:	T_MaxString; // \\PC-Name\Folder\ C:\Folder\
	File													:	STRING := '*.*'; // *.xml / *.txt
END_VAR
VAR_OUTPUT
	NoOfFiles												:	INT; //Number of files found in folder and sub folder
	EoE														:	BOOL; //end of enumeration - No more files in folder
	Entrys													:	ARRAY[MIN_ENTRYS..MAX_ENTRYS] OF ST_FindFileEntry; //List of file structures
END_VAR
VAR
(* internal used variables ************************************************************)
	
(* trigger ****************************************************************************)	

(* function-block instances ***********************************************************)
	EnumFindFileEntry										:	FB_EnumFindFileEntry;
END_VAR


(* Sequence ****************************************)
	rtExecute(CLK := Execute);
	CASE state OF 
	0:	
		Busy												:= FALSE;
		IF NOT Execute
		THEN
			Done											:= FALSE;
			Error											:= FALSE;
			ErrorId											:= 0;
		ELSIF rtExecute.Q
		THEN
			EnumFindFileEntry(bExecute := FALSE, sNetId := AMSNetId, tTimeout := Timeout, sPathName := CONCAT(Path,File));
			Busy											:= TRUE;
			Done											:= FALSE;
			Error											:= FALSE;
			ErrorId											:= 0;
			NoOfFiles										:= 0;
			MEMSET(ADR(Entrys),0,SIZEOF(Entrys));
			state											:= State + 1;
		END_IF 
	
	1: //read first entry
		EnumFindFileEntry(bExecute := TRUE ,eCmd := eEnumCmd_First );
		state												:= State + 1;

	2: //read entrys
		EnumFindFileEntry(bExecute := TRUE);
		IF NOT EnumFindFileEntry.bBusy
		THEN
			IF NOT EnumFindFileEntry.bError
			THEN
				IF EnumFindFileEntry.bEOE		
				THEN
					Busy									:= FALSE;
					Done									:= TRUE;	
					state									:= 0;
					
				ELSIF NOT EnumFindFileEntry.stFindFile.fileAttributes.bDirectory
				THEN
					NoOfFiles								:= LIMIT(MIN_ENTRYS, NoOfFiles + 1 ,MAX_ENTRYS);
					Entrys[NoOfFiles]						:= EnumFindFileEntry.stFindFile;
					
					IF EnumFindFileEntry.bEOE
					THEN
						EoE									:= TRUE;
						Busy								:= FALSE;
						Done								:= TRUE;
						state								:= 0;
					ELSIF NoOfFiles >= MAX_ENTRYS
					THEN
						state								:= 3;
					ELSE
						; //Continue with next cycle					
					END_IF		
					
				END_IF
				EnumFindFileEntry(bExecute := FALSE ,eCmd := eEnumCmd_Next);
			ELSE
				Busy										:= FALSE;
				Done										:= FALSE;
				Error										:= TRUE;
				ErrorId										:= EnumFindFileEntry.nErrID;
				state										:= 0;
			END_IF		
		END_IF
		
	3: //End search
		EnumFindFileEntry(bExecute := TRUE ,eCmd := eEnumCmd_Abort);
		IF NOT EnumFindFileEntry.bBusy
		THEN
			Busy											:= FALSE;
			Done											:= NOT EnumFindFileEntry.bError;
			Error											:= NOT Done;
			ErrorId											:= EnumFindFileEntry.nErrID;
			state											:= 0;		
		END_IF
	
	END_CASE

(*************************************************************************)

END_FUNCTION_BLOCK

// ---- POUs/IO/Analog/AnalogIn.TcPOU
{attribute 'no_check'}
FUNCTION_BLOCK AnalogIn
VAR_INPUT
	MinValue												: 	LREAL 	:= 0.0; //In case of extended range (107%), set Options.5 or MinValue accordingly e.g. -10.7V (instead of -10.0V as scaling is based on full 16bit)
	MaxValue												: 	LREAL 	:= 0.0; //In case of extended range (107%), set Options.5 or MaxValue accordingly e.g. 10.7V (instead of 10.0V as scaling is based on full 16bit)
	NoOfDigits												: 	INT 	(0..10)	:= 0; 	//number of decimal digits of scaled Q variable 
	OutOnError												:	LREAL 	:= 0.000000000000000001;
{attribute 'displaymode':='binary'}                     	
	Options													:	BYTE  := 2#0000_0000; (* 	.0 = FALSE scale value from 0 <-> 32767 / TRUE scale value with sign -32768 <-> 32767
																							.4 = Active only if .0 AND .5 =TRUE | FALSE scale value min -32768 / TRUE scale value changed from -30518 to -7629 -> Ext. Range Mode of e.g. 4-20mA where 0mA is equel -7629 
																							.5 = FALSE legacy range with FSV OF 100%=+-32767 / TRUE TO enable extended range AND applying ~7% TO MIN/MaxValue (with ext. range act. measurement can be exceeded OR undershot BY approx. 7% setting FSV TO 100%=+/-30518 AND 107% representing full 16BIT) 
																							For Scaling of 4-20mA according to NAMUR bit .0,.4 and .5 have to be set *)

																							
	Offset													:	LREAL := 0.0;
END_VAR                 									
VAR                                                     	
END_VAR                                                 	
VAR_OUTPUT                                              	
	Q														:	LREAL;		//Scaled result value
	In											AT  %I* 	: 	INT; 		//Hardware Input

{attribute 'displaymode':='binary'}                     	
	Status										AT  %I*		:	WORD := 2#0000_0000_0000_0000; //Terminal status word -> can also be linked with status byte 
END_VAR
VAR
END_VAR

(* read analog value 																					   *)
(* resolution process image			e.g.							/ 0V = 0 / 10V = 32767 / -10V = -32768 *)
(* or directly with NoOfDigits																	250 -> 25.0°*)
(************************************************************************************************************)
	
(* Scaling ******************************************************************)
	IF MaxValue <> MinValue 
	THEN
		Q 													:= Offset + scale2(In , SEL(Options.0, 0.0, SEL(Options.5 , -32768.0, SEL(Options.4, -30518.0,-7629.0) ) ), SEL(Options.5,32767.0,30518.0), MinValue, MaxValue);
		IF NoOfDigits > 0
		THEN
			Q												:= TO_FMLREAL(Q,NoOfDigits);
		END_IF
	
	ELSIF NoOfDigits > 0 (* Bsp PT100 *)
	THEN
		Q													:= Offset + TO_FMLREAL(In,NoOfDigits);
		
	ELSE  													
		Q 													:= 0.0;
	END_IF

	IF 	Error AND OutOnError <> 0.000000000000000001
	THEN
		Q													:= OutOnError;
	END_IF
(**********************************************************************************************************************)

{attribute 'monitoring' := 'call'}
PROPERTY PUBLIC Error : BOOL
GET
Error					:= Status.6 OR MinValue = MaxValue AND NoOfDigits = 0;
END_GET
END_PROPERTY

{attribute 'monitoring' := 'call'}
PROPERTY PUBLIC Limit_1 : BYTE
GET
Limit_1.0					:= Status.2;
Limit_1.1					:= Status.3;
END_GET
END_PROPERTY

{attribute 'monitoring' := 'call'}
PROPERTY PUBLIC Limit_2 : BYTE
GET
Limit_2.0					:= Status.4;
Limit_2.1					:= Status.5;
END_GET
END_PROPERTY

PROPERTY PUBLIC optEnableScaleExtRangeMode : bool
GET
optEnableScaleExtRangeMode := Options.5;
END_GET
SET
Options.5 := optEnableScaleExtRangeMode;
END_SET
END_PROPERTY

PROPERTY PUBLIC optEnableScaleExtRangeModeNeg7629 : bool
GET
optEnableScaleExtRangeModeNeg7629 := Options.4;
END_GET
SET
Options.4 := optEnableScaleExtRangeModeNeg7629;
END_SET
END_PROPERTY

PROPERTY PUBLIC optEnableScaleSignedValue : bool
GET
optEnableScaleSignedValue := Options.0;
END_GET
SET
Options.0 := optEnableScaleSignedValue;
END_SET
END_PROPERTY

{attribute 'monitoring' := 'call'}
PROPERTY PUBLIC Overrange : BOOL
GET
Overrange					:= Status.1;
END_GET
END_PROPERTY

{attribute 'monitoring' := 'call'}
PROPERTY PUBLIC SyncError : BOOL
GET
SyncError 			:= Status.13;
END_GET
END_PROPERTY

{attribute 'monitoring' := 'call'}
PROPERTY PUBLIC TxPDOState : BOOL
GET
TxPDOState					:= Status.14; //True if not valid
END_GET
END_PROPERTY

{attribute 'monitoring' := 'call'}
PROPERTY PUBLIC TxPDOToggle : BOOL
GET
TxPDOToggle						:= Status.15;
END_GET
END_PROPERTY

{attribute 'monitoring' := 'call'}
PROPERTY PUBLIC Underrange : BOOL
GET
Underrange 					:= Status.0;
END_GET
END_PROPERTY

END_FUNCTION_BLOCK

// ---- POUs/IO/Analog/AnalogIn32.TcPOU
{attribute 'no_check'}
FUNCTION_BLOCK AnalogIn32 extends EcSlaveInfoDataExt
VAR_INPUT
	MinValue												: 	LREAL 	:= 0.0;
	MaxValue												: 	LREAL 	:= 0.0;
	NoOfDigits												: 	INT 	(0..10)	:= 0; //number of decimal digits of scaled Q variable 
	OutOnError												:	LREAL 	:= 0.000000000000000001;
{attribute 'displaymode':='binary'}     	            	
	Options													:	BYTE  := 2#0000_0010; (* .0 = FALSE Scale value from 0 to e.g. 32767 / TRUE scale singed value e.g. -32768 <-> 32767 , see Options .1 and .2 for more scaling Options 
																						.1 = FALSE = 32 bit resolution / TRUE = value is based on 24 bit resolution e.g. -> -8388608.0 or 0.0 <-> 8388607.0 
																						.2 = Right adjust of 32/24 bit value -> value will be shifted by 8 bits (divided bv 256)   
																						.3 = TRUE = Enable extended range mode -> change scaling to +/-7812500 instead of r+/- 838860x *)
	Offset													:	LREAL := 0.0;
END_VAR                 									                                	            	
VAR_OUTPUT                              	            	
	Q														:	LREAL;	//scaled result value
	In											AT  %I* 	: 	DINT; 	//Hardware Input 
{attribute 'displaymode':='binary'}     	            	
	Status										AT  %I*		:	WORD := 2#0100_0000_0000_0000;	//Terminal status word -> can also be linked with status byte
END_VAR

(* read 32bit analog value 																				    *)
(* resolution process image			e.g.				/ 0V = 0 / 10V = 2147483647 / -10V = - 2147483647 	*)
(* or directly with NoOfDigits																	250 -> 25.0°*)
(************************************************************************************************************)
	
(* Scaling ******************************************************************)
	IF MaxValue <> MinValue 
	THEN
		IF Options.1 
		THEN //24 bit resolution
			IF NOT Options.3
			THEN
				Q 	 										:= Offset + scale(SEL(Options.2 , In , In / 256.0 ) , SEL(Options.0, 0.0, -8388608.0), 8388607.0, MinValue , MaxValue);
			ELSE
		 		Q 	 										:= Offset + scale(SEL(Options.2 , In , In / 256.0 ) , SEL(Options.0, 0.0, -7812500.0), 7812500.0, MinValue , MaxValue);
			END_IF
		ELSE //32 bit resolution 
			Q 	 											:= Offset + scale(SEL(Options.2 , In , In / 256.0 ) , SEL(Options.0, 0.0, -2147483648.0), 2147483647.0, MinValue , MaxValue);		
		END_IF
		IF NoOfDigits > 0
		THEN
			Q												:= TO_FMLREAL(Q,NoOfDigits);
		END_IF
	
	ELSIF NoOfDigits > 0 (* Bsp PT100 *)
	THEN
		Q													:= Offset + TO_FMLREAL(In,NoOfDigits);
		
	ELSE  													
		Q 													:= 0.0;
	END_IF

	IF 	Error AND OutOnError <> 0.000000000000000001
	THEN
		Q													:= OutOnError;
	END_IF
(**********************************************************************************************************************)

{attribute 'monitoring' := 'call'}
PROPERTY PUBLIC Error : BOOL
GET
Error					:= Status.6 OR MinValue = MaxValue AND NoOfDigits = 0;
END_GET
END_PROPERTY

{attribute 'monitoring' := 'call'}
PROPERTY PUBLIC Limit_1 : BYTE
GET
Limit_1.0					:= Status.2;
Limit_1.1					:= Status.3;
END_GET
END_PROPERTY

{attribute 'monitoring' := 'call'}
PROPERTY PUBLIC Limit_2 : BYTE
GET
Limit_2.0					:= Status.4;
Limit_2.1					:= Status.5;
END_GET
END_PROPERTY

PROPERTY optEnable24BitResolution : BOOL //In value is provided as 32bit value instead if 24bit
GET
optEnable24BitResolution := Options.1;
END_GET
SET
Options.1 := optEnable24BitResolution;
END_SET
END_PROPERTY

PROPERTY PUBLIC optEnableScaleExtRangeMode : bool
GET
optEnableScaleExtRangeMode := Options.3;
END_GET
SET
Options.3 := optEnableScaleExtRangeMode;
END_SET
END_PROPERTY

PROPERTY PUBLIC optEnableScaleSignedValue : bool
GET
optEnableScaleSignedValue := Options.0;
END_GET
SET
Options.0 := optEnableScaleSignedValue;
END_SET
END_PROPERTY

PROPERTY PUBLIC optShiftValueBy8Bits : BOOL
GET
optShiftValueBy8Bits := Options.2;
END_GET
SET
Options.2 := optShiftValueBy8Bits;
END_SET
END_PROPERTY

{attribute 'monitoring' := 'call'}
PROPERTY PUBLIC Overrange : BOOL
GET
Overrange					:= Status.1;
END_GET
END_PROPERTY

{attribute 'monitoring' := 'call'}
PROPERTY PUBLIC SyncError : BOOL
GET
SyncError 			:= Status.13;
END_GET
END_PROPERTY

{attribute 'monitoring' := 'call'}
PROPERTY PUBLIC TxPDOState : BOOL
GET
TxPDOState					:= Status.14; //True if not valid
END_GET
END_PROPERTY

{attribute 'monitoring' := 'call'}
PROPERTY PUBLIC TxPDOToggle : BOOL
GET
TxPDOToggle						:= Status.15;
END_GET
END_PROPERTY

{attribute 'monitoring' := 'call'}
PROPERTY PUBLIC Underrange : BOOL
GET
Underrange 					:= Status.0;
END_GET
END_PROPERTY

END_FUNCTION_BLOCK

// ---- POUs/_Miscellaneous/scale.TcPOU
//Discription:	"SCALE" scales the In-Value in the range between InLow to InHigh, to the commited OutLow to OutHigh range (In will be limited by InLow/InHigh).
//Used for AnalogIn/Out
FUNCTION scale : LREAL
VAR_INPUT
	In				 										: LREAL;
	InLow 													: LREAL;
	InHigh 													: LREAL;
	OutLow 													: LREAL;
	OutHigh 												: LREAL;
END_VAR
VAR
	Lim														: LREAL;
	X														: LREAL;
END_VAR

IF OutHigh <> OutLow 
THEN
	X														:= InHigh - InLow;
	IF x <> 0.0             									
	THEN       
		Lim 												:= LIMIT(InLow,In,InHigh) - InLow;             									
		X		 											:= (OutHigh - OutLow) / X;
		scale 												:= (X * Lim) + OutLow;			
	ELSE                    									
		scale												:= 0.0;
	END_IF
ELSE
	scale													:= 0.0;	
END_IF

END_FUNCTION

// ---- POUs/IO/Analog/AnalogInELMSingleSampleDINT.TcPOU
// AnalogIn FB to read and scale a single DINT (24bit) sample input from ELMxxxx terminal
// Set bit 3 (Options.3) to true to enable scaling based on +/-7812500 instead of legacy range values +/-838860x
FUNCTION_BLOCK AnalogInELMSingleSampleDINT EXTENDS AnalogInELMBase
VAR_INPUT
	Offset													:	LREAL := 0.0;

END_VAR                 									
VAR                                     	            	
END_VAR                                 	            	
VAR_OUTPUT                              	            	                                       	
	Q														:	LREAL;	//scaled result value
	In											AT  %I* 	: 	DINT; 	//Hardware Input 
END_VAR                                 	
VAR                                   	
END_VAR

(* Read single DINT sample value from ELM terminal and scale to user units									*)
(************************************************************************************************************)

(* evaluate statusword **************************************************************************************)
	SUPER^();
	
(* Scaling ******************************************************************)
	IF MaxValue <> MinValue 
	THEN	
		IF NOT Options.3
		THEN
			Q 	 											:= Offset + Scale(TO_LREAL(In) , -8388608.0, 8388607.0, MinValue , MaxValue);
		ELSE
			Q 	 											:= Offset + Scale(TO_LREAL(In), -7812500.0, 7812500.0, MinValue , MaxValue);
		END_IF	
		IF NoOfDigits > 0
		THEN
			Q												:= TO_FMLREAL(Q,NoOfDigits);
		END_IF
	
	ELSIF NoOfDigits > 0 (* Bsp PT100 *)
	THEN
		Q													:= Offset + TO_FMLREAL(In,NoOfDigits);
		
	ELSE  													
		Q 													:= 0.0;
	END_IF

	IF 	Error AND OutOnError <> 0.000000000000000001
	THEN
		Q													:= OutOnError;
	END_IF
(**********************************************************************************************************************)

METHOD FB_init : BOOL
VAR_INPUT
	bInitRetains : BOOL; // if TRUE, the retain variables are initialized (warm start / cold start)
	bInCopyCode : BOOL;  // if TRUE, the instance afterwards gets moved into the copy code (online change)
END_VAR
IF NOT bInCopyCode THEN
	NoOfDigits 							:= 2;
END_IF
END_METHOD

PROPERTY PUBLIC optEnableScaleExtRangeMode : bool
GET
optEnableScaleExtRangeMode := Options.3;
END_GET
SET
Options.3 := optEnableScaleExtRangeMode;
END_SET
END_PROPERTY

END_FUNCTION_BLOCK

// ---- POUs/IO/Analog/AnalogInREAL.TcPOU
// AnalogInReal FB to read and scale a single REAL input
// Set bit 3 (Options.3) to true to enable scaling based on +/-7812500 instead of legacy range values +/-838860x
// NoOfDigits per default set to 3... 
FUNCTION_BLOCK AnalogInREAL EXTENDS EcSlaveInfoDataExt
VAR_INPUT
	Offset													:	LREAL 		:= 0.0;
	MinValue												: 	LREAL 		:= 0.0;
	MaxValue												: 	LREAL 		:= 0.0;
	NoOfDigits												: 	INT(0..10)	:= 0; //number of decimal digits of scaled Q variable 
	OutOnError												:	LREAL 		:= 0.000000000000000001;
{attribute 'displaymode':='binary'}     	            	
	Options													:	BYTE  		:= 2#0000_0000;
END_VAR                 									
VAR                        
END_VAR                                 	            	
VAR_OUTPUT                              	            	                                       	
	Q														:	LREAL;//scaled result value
	In											AT  %I* 	: 	REAL; //Hardware Input
	{attribute 'displaymode':='binary'}     	            	
	Status										AT  %I*		:	WORD := 2#00000000_00000000;	//Terminal status (2 bytes)
END_VAR

(* Read single REAL value from terminal and scale to user units				*)
(****************************************************************************)

(* Scaling ******************************************************************)
	IF MaxValue <> MinValue 
	THEN			
		IF NOT Options.3
		THEN
			Q 	 											:= Offset + Scale(TO_LREAL(In), -8388608.0, 8388607.0, MinValue , MaxValue);
		ELSE
			Q 	 											:= Offset + Scale(TO_LREAL(In),  -7812500.0, 7812500.0, MinValue , MaxValue);		
		END_IF	
		
		IF NoOfDigits > 0
		THEN
			Q												:= TO_FMLREAL(Q,NoOfDigits);
		END_IF
	
	ELSIF NoOfDigits > 0 (* Bsp PT100 *)
	THEN
		Q													:= Offset + TO_FMLREAL(In,NoOfDigits);
		
	ELSE  													
		Q 													:= 0.0;
	END_IF

(****************************************************************************)

{attribute 'monitoring' := 'call'}
PROPERTY PUBLIC Error : BOOL
GET
Error					:= Status.6 OR MinValue = MaxValue AND NoOfDigits = 0;
END_GET
END_PROPERTY

{attribute 'monitoring' := 'call'}
PROPERTY PUBLIC Limit_1 : BYTE
GET
Limit_1.0					:= Status.2;
Limit_1.1					:= Status.3;
END_GET
END_PROPERTY

{attribute 'monitoring' := 'call'}
PROPERTY PUBLIC Limit_2 : BYTE
GET
Limit_2.0					:= Status.4;
Limit_2.1					:= Status.5;
END_GET
END_PROPERTY

PROPERTY PUBLIC optEnableScaleExtRangeMode : bool
GET
optEnableScaleExtRangeMode := Options.3;
END_GET
SET
Options.3 := optEnableScaleExtRangeMode;
END_SET
END_PROPERTY

{attribute 'monitoring' := 'call'}
PROPERTY PUBLIC Overrange : BOOL
GET
Overrange 			:= Status.1;
END_GET
END_PROPERTY

{attribute 'monitoring' := 'call'}
PROPERTY PUBLIC TareActive : BOOL
GET
TareActive					:= Status.11;
END_GET
END_PROPERTY

{attribute 'monitoring' := 'call'}
PROPERTY PUBLIC TxPDOState : BOOL
GET
TxPDOState					:= Status.14; //True if not valid
END_GET
END_PROPERTY

{attribute 'monitoring' := 'call'}
PROPERTY PUBLIC TxPDOToggle : BOOL
GET
TxPDOToggle							:= Status.15;
END_GET
END_PROPERTY

{attribute 'monitoring' := 'call'}
PROPERTY PUBLIC Underrange : BOOL
GET
Underrange 			:= Status.0;
END_GET
END_PROPERTY

END_FUNCTION_BLOCK

// ---- POUs/IO/Button.TcPOU
{attribute 'no_check'}
FUNCTION_BLOCK Button 
VAR_INPUT
	Enable													:	BOOL := TRUE;	//FB will be processed as long as enable is TRUE 
	Force													:	BOOL := FALSE; 	//simulates Input signal
	Invert													:	BOOL := FALSE; 	//inverts the Hardware Input
	LED												AT  %Q*	:	BOOL;			//LED/Light hardware output
END_VAR         									
VAR_OUTPUT
	Q														:	BOOL;	//direct signal
	Q_RT													:	BOOL;	//R_Trig signal of delay Q
	Q_FT													:	BOOL;	//F_Trig signal of delay Q
	Q_TGL													:	BOOL;	//Toggle -> use flag Q_RT
	In												AT  %I*	:	BOOL; 	//Hardware Input
END_VAR
VAR
	Mem														:	BOOL;
END_VAR

(* Taster mit Togglefunktion V1.0						*)
(********************************************************)

(********************************************************)
Mem															:= Q;
Q 															:= ((In OR Force) XOR Invert) AND Enable;
Q_RT 														:= NOT Mem AND Q;
Q_FT														:= Mem AND NOT Q;
Q_TGL 														:= (Q_RT XOR Q_TGL);
(********************************************************)

METHOD PUBLIC setDisable : BOOL
VAR_INPUT
END_VAR
Enable 														:= FALSE;
setDisable													:= TRUE;
END_METHOD

METHOD PUBLIC setEnable : bool
VAR_INPUT
END_VAR
Enable 														:= TRUE;
setEnable													:= TRUE;
END_METHOD

METHOD PUBLIC setLedOFF : bool
VAR_INPUT
END_VAR
LED 														:= FALSE;
setLEDOff													:= TRUE;
END_METHOD

METHOD PUBLIC setLedON : booL
VAR_INPUT
END_VAR
LED 														:= TRUE;
setLedON													:= TRUE;
END_METHOD

METHOD PUBLIC TGL : booL //Return value = Q_TGL status
VAR_INPUT
END_VAR
TGL := Q_TGL 														:= NOT Q_TGL;
END_METHOD

METHOD PUBLIC TglOff : booL
VAR_INPUT
END_VAR
Q_TGL 														:= FALSE;
TglOFF														:= TRUE;
END_METHOD

METHOD PUBLIC TglOn : bool
VAR_INPUT
END_VAR
Q_TGL 														:= TRUE;
TglON														:= TRUE;
END_METHOD

END_FUNCTION_BLOCK

// ---- POUs/IO/Cylinder/Cylinder.TcPOU
{attribute 'no_check'}
//Cylinder object with two outputs (Workpos./Basepos) and correlated inputs
//Via the Options byte, it is possible to disable the use either of one or both feedback inputs.
//In case the physical feedback input in disabled, the status output of the FB will be generated by PT_Feedback
//In case the physical feedback input will not be triggerd to his corresonding outout within a certain time (PT_Feedback), an timeout error occures
//The physical outputs could be blocked by set the FeedxxxPos signals to false.
//FB "INPUT" is used inside
FUNCTION_BLOCK Cylinder IMPLEMENTS I_Cylinder
VAR_OUTPUT CONSTANT
{attribute 'displaymode':='binary'}
	OPTION_DISABLE_SENSOR_BASEPOS							:	BYTE  := 2#0000_0001; //Disable sensor check basepos. Feedback time used instead to create signal
{attribute 'displaymode':='binary'}
	OPTION_DISABLE_SENSOR_WORKPOS							:	BYTE  := 2#0000_0010; //Disable sensor check workpos. Feedback time used instead to create signal
{attribute 'displaymode':='binary'}
	OPTION_FREE												:	BYTE  := 2#0000_0100; //Not used option		
{attribute 'displaymode':='binary'}
	OPTION_DISABLE_LOGIC_ERROR								:	BYTE  := 2#0000_1000; //Disable logic error (Sensor workpos and basepos active at the same time) 	
{attribute 'displaymode':='binary'}
	OPTION_SWAP_SENSOR_STATUS								:	BYTE  := 2#0001_0000; //Swap signals work and base pos at Status byte
{attribute 'displaymode':='binary'}
	OPTION_INVERT_SENSOR_BASEPOS							:	BYTE  := 2#0010_0000; //Invert logic of sensor basepos (->NO)
{attribute 'displaymode':='binary'}
	OPTION_INVERT_SENSOR_WORKPOS							:	BYTE  := 2#0100_0000;//Invert logic of sensor workpos (->NO)
{attribute 'displaymode':='binary'}
	OPTION_EN_IMPULS_VALVE									:	BYTE  := 2#1000_0000; //Outputs are switched off if endposition is reached	
END_VAR
VAR_INPUT  (* Peripherie Outputs *)
	Quit													:	BOOL;	//Resets error with rising edge
	ToWorkPos												:	BOOL;	//moves cylinder to work position
	ToBasePos												:	BOOL;	//moves cylinder to base position
{attribute 'displaymode':='binary'}         			
	Options													:	BYTE  := 2#0000_0000;  (* option constants are predefined, so they can accordingly be passed symbolically to the block
																							DISABLE_FEEDBACK_BP	= .0
																							DISABLE_FEEDBACK_WP	= .1
																							ENABLE_LATCH_ERROR	= .2
																							DISABLE_LOGIC_ERROR	= .3																							
																							SWAP_SENSOR_STATUS	= .4
																							FEEDBACK_BP_INVERT	= .5
																							FEEDBACK_WP_INVERT	= .6
																							IMPULS_VALVE		= .7
																									*)
	FeedBasePos												:	BOOL := TRUE;	//enables feed in base direction
	FeedWorkPos												:	BOOL := TRUE;	//enables feed in work direction
	PT_Timeout												:	TIME := T#5S; 	//Runtime check BasePos
	PT_Feedback												:	TIME := T#3S; 	//Delay simulate Feedback
	PT_SensorDamping										:	TIME := T#0MS; 	//Work and Base pos sensor on/off damping time to suppress sensor flickering  
END_VAR                                     			
VAR_OUTPUT  (* Peripherie Inputs *)         			
	InBasePos												:	BOOL;	//TRUE when cylinder is in base position
	InWorkPos												:	BOOL;	//TRUE when cylinder is in work position
	Done													:	BOOL; 	//Limit sensor reached or feedback time counted down
	Busy													:	BOOL;	//Busy is TRUE at the rising edge of Execute and FALSE when one of the outputs Done, Aborted, or Error is set 
	ErrBasePos												:	BOOL;	//Cannot reach base position
	ErrWorkPos												:	BOOL;	//Cannot reach work position  
	ErrLogic												:	BOOL; 	//Both feedback signals are on
{attribute 'displaymode':='binary'}         			
	Status													:	BYTE;	(* 	Bit 0 = Q_ToBasePos or opposite if status swap in Options is active
																			Bit 1 = Q_ToWorkPos or opposite if status swap in Options is active
																			Bit 2 = InBasePos or opposite if status swap in Options is active
																			Bit 3 = InWorkPos or opposite if status swap in Options is active
																			Bit 4 = FeedBasePos or opposite if status swap in Options is active
																			Bit 5 = FeedWorkPos or opposite if status swap in Options is active
																			Bit 6 = Ready (no error)
																			Bit 7 = Error timeout move to position or sensor logic
																		*)
	Q_ToBasePos										AT  %Q* :	BOOL; //Hardware output - only with read access
	Q_ToWorkPos										AT  %Q* :	BOOL; //Hardware output - only with read access
END_VAR
VAR// IOs 
	SensorBasePos											: INPUT;
	SensorWorkPos											: INPUT;	
	TonErrBasePos											: TON;
	TonErrWorkPos											: TON;
	SimulationOn											:	BOOL;
END_VAR

	(* Cylinder	 IO V2.9					 								       	*)
	(* Includes functionblock "INPUT" 												*)
	(********************************************************************************)

(* Write Output *****************************************************)
	IF ToBasePos 	
	THEN
		moveToBasePos();
	ELSIF ToWorkPos AND NOT ToBasePos
	THEN
		moveToWorkPos();
	ELSE
		switchOff();
	END_IF

(* Reedkontakte lesen ***********************************************)
	this^._readSensors();
	
(* Status *************************************************)
	_writeStatus();
                        	
(* ack Error **********************************************************)
	IF Quit  THEN  reset(); END_IF

(* Timeout  ************************************************)
	_runtimeChk();
	
(*********************************************************************)

METHOD PROTECTED _readSensors : BOOL
VAR_INPUT
END_VAR
	SensorBasePos(
		Force	:= Q_ToBasePos AND NOT InWorkPos AND(Options.0 OR SimulationOn),
		Invert	:= Options.5,
		PT_ON	:= SEL(Options.0 OR SimulationOn,PT_SensorDamping,PT_FEEDBACK),
		PT_OFF	:= SEL(Options.0 OR SimulationOn,PT_SensorDamping,T#0MS),
		Q_DIRECT=>,
		Q		=> InBasePos,
		Q_RT	=> ,
		Q_FT	=> ,
		IN		=> );


	SensorWorkPos(
		Force	:= Q_ToWorkPos AND NOT InBasePos AND(Options.1 OR SimulationOn),
		Invert	:= Options.6,
		PT_ON	:= SEL(Options.1 OR SimulationOn ,PT_SensorDamping,PT_FEEDBACK),
		PT_OFF	:= SEL(Options.1 OR SimulationOn ,PT_SensorDamping,T#0MS),
		Q_DIRECT=>,
		Q		=> InWorkPos,
		Q_RT	=> ,
		Q_FT	=> ,
		IN		=> );
		

	_readSensors									:= TRUE;
END_METHOD

METHOD PROTECTED _runtimeChk : BOOL
VAR_INPUT
END_VAR
(* Timeout WorkPos ************************************************)
	TonErrWorkPos(	IN := Q_ToWorkPos AND (NOT InWorkPos OR InBasePos),
					PT := MAX(PT_Timeout + PT_SensorDamping,PT_Feedback + T#1S),
					Q => ErrWorkPos);

(* Timeout WorkPos ************************************************)
	tonErrBasePos(	IN := Q_ToBasePos AND (NOT InBasePos OR InWorkPos),
					PT := MAX(PT_Timeout + PT_SensorDamping,PT_Feedback + T#1S),
					Q => ErrBasePos);
					
(*********************************************************************)
	_runtimeChk									:= TRUE;
END_METHOD

METHOD PROTECTED _writeStatus : BOOL
VAR_INPUT
END_VAR


	(* Move *)
	IF Q_ToBasePos AND NOT Q_ToWorkPos AND (NOT InBasePos OR InWorkPos)
	THEN
		Status.0 											:= NOT Options.4;
		Status.1											:= Options.4;
	ELSIF Q_ToWorkPos AND NOT Q_ToBasePos AND (NOT InWorkPos OR InBasePos)
	THEN
		Status.0											:= Options.4;
		Status.1											:= NOT Options.4;
	END_IF              									

	(* BasePos / WorkPos reached*)
	Status.2 												:= SEL(Options.4, InBasePos , InWorkPos);
	Status.3 												:= SEL(Options.4, InWorkPos , InBasePos);
 				        									
	(* Feed ok *)    									
	Status.4 												:= SEL(Options.4, FeedBasePos , FeedWorkPos);
	Status.5 												:= SEL(Options.4, FeedWorkPos , FeedBasePos);
                        									
	(* Ready *)         									
	Status.6												:= NOT Status.7; 
	                    									
	(* Error *)         									
	Status.7 												:= ErrBasePos OR ErrWorkPos OR ErrLogic;
	
	(* Logic error bit **********************************************)
	ErrLogic												:= InBasePos AND InWorkPos AND NOT Options.3;
	
	(* Result *)
	_writeStatus												:= TRUE;
END_METHOD

METHOD PUBLIC enable : BOOL //Return Done = TRUE if WorkPos is TRUE and InWorkPos = TRUE or WorkPos is FALSE and InBasePos is TRUE 
VAR_INPUT
	IN													:	BOOL; //TRUE=WORK / FALSE=BASE
END_VAR
IF IN
THEN
	Enable 													:= THIS^.moveToWorkPos();
ELSE
	Enable 													:= This^.moveToBasePos();
END_IF
END_METHOD

{attribute 'monitoring' := 'call'}
PROPERTY PUBLIC inError : Bool
GET
InError									:= Status.7;
END_GET
END_PROPERTY

{attribute 'monitoring' := 'call'}
PROPERTY public isBusy : bool
GET
isBusy := Busy;
END_GET
END_PROPERTY

{attribute 'monitoring' := 'call'}
PROPERTY isInBasePos : BOOL
GET
isInBasePos := InBasePos;
END_GET
END_PROPERTY

{attribute 'monitoring' := 'call'}
PROPERTY isInWorkPos : BOOL
GET
isInWorkPos := InWorkPos;
END_GET
END_PROPERTY

{attribute 'monitoring' := 'call'}
PROPERTY public isOff : BOOL
GET
isOff := not ToWorkPos and not ToBasePos;
END_GET
END_PROPERTY

METHOD PUBLIC moveToBasePos : BOOL //Return = Done -> InBasePos
ToWorkPos 									:= Q_ToWorkPos	:= FALSE;
ToBasePos 													:= TRUE;
Q_ToBasePos	 												:= FeedBasePos AND (NOT Options.7 OR NOT InBasePos);
moveToBasePos 									:= Done			:= InBasePos;
Busy														:= NOT Done;
END_METHOD

METHOD PUBLIC moveToWorkPos : BOOL //Return = Done -> InWorkPos
ToBasePos 								:= Q_ToBasePos 		:= FALSE;
ToWorkPos													:= TRUE;
Q_ToWorkPos	 												:= FeedWorkPos AND (NOT Options.7 OR NOT InWorkPos);
moveToWorkPos								:= Done 				:= InWorkPos;
Busy														:= NOT Done;
END_METHOD

{attribute 'monitoring' := 'call'}
PROPERTY PUBLIC noFeed : BOOL
GET
noFeed						:= ToWorkPos and not FeedWorkPos or ToBasePos and not FeedBasePos;
END_GET
END_PROPERTY

{attribute 'monitoring' := 'call'}
PROPERTY Public ok : bool
GET
ok := Done;
END_GET
END_PROPERTY

{attribute 'monitoring' := 'call'}
PROPERTY PUBLIC optDisableLogicError : BOOL
GET
optDisableLogicError := Options.3;
END_GET
SET
Options.3 := optDisableLogicError;
END_SET
END_PROPERTY

{attribute 'monitoring' := 'call'}
PROPERTY PUBLIC optDisableSensorBasepos : BOOL
GET
optDisableSensorBasepos := Options.0;
END_GET
SET
OPtions.0 := optDisableSensorBasepos;
END_SET
END_PROPERTY

{attribute 'monitoring' := 'call'}
PROPERTY PUBLIC optDisableSensorWorkpos : BOOL
GET
optDisableSensorWorkpos := Options.1;
END_GET
SET
OPtions.1 := optDisableSensorWorkpos;
END_SET
END_PROPERTY

{attribute 'monitoring' := 'call'}
PROPERTY PUBLIC optEnableImpulsValveFnc : BOOL
GET
optEnableImpulsValveFnc := Options.7;
END_GET
SET
Options.7 := optEnableImpulsValveFnc;
END_SET
END_PROPERTY

{attribute 'monitoring' := 'call'}
PROPERTY PUBLIC optInvertSensorBasepos : BOOL
GET
optInvertSensorBasepos := Options.5;
END_GET
SET
Options.5 := optInvertSensorBasepos;
END_SET
END_PROPERTY

{attribute 'monitoring' := 'call'}
PROPERTY PUBLIC optInvertSensorWorkpos : BOOL
GET
optInvertSensorBasepos := Options.6;
END_GET
SET
Options.6 := optInvertSensorBasepos;
END_SET
END_PROPERTY

{attribute 'monitoring' := 'call'}
PROPERTY PUBLIC optSwapSensorStatus : BOOL
GET
optSwapSensorStatus := Options.4;
END_GET
SET
OPtions.4 := optSwapSensorStatus;
END_SET
END_PROPERTY

{attribute 'monitoring' := 'call'}
PROPERTY PUBLIC rCylinder : REFERENCE TO Cylinder
GET
rCylinder REF= This^;
END_GET
END_PROPERTY

METHOD PUBLIC reset : BOOL //Result = reset done
	TonErrWorkPos(IN := FALSE);
	tonErrBasePos(IN := FALSE);
	ErrWorkPos	:= ErrBasePos := ErrLogic						:= FALSE;										
	Status.7 													:= FALSE;
	reset														:= TRUE;
END_METHOD

{attribute 'monitoring' := 'call'}
PROPERTY simulation : BOOL
GET
simulation := SimulationOn;
END_GET
SET
SimulationOn := simulation;
END_SET
END_PROPERTY

METHOD PUBLIC switchOff : BOOL
VAR_INPUT
END_VAR
	ToWorkPos	:= FALSE;
	ToBasePos	:= FALSE;
	Done		:= FALSE;
	Busy		:= FALSE;
	Q_ToBasePos	:= FALSE;
	Q_ToWorkPos	:= FALSE;
	switchOff	:= TRUE;
END_METHOD

END_FUNCTION_BLOCK

// ---- POUs/IO/Cylinder/CylinderType4.TcPOU
{attribute 'no_check'}
//Cylinder with 2x inputs each for work and base position, extended from FB Cylinder
FUNCTION_BLOCK CylinderType4 EXTENDS Cylinder
VAR_OUTPUT CONSTANT
END_VAR
VAR_INPUT  
END_VAR                                     			
VAR_OUTPUT    
{attribute 'displaymode':='binary'}
	ErrInfo													:	BYTE; //.0 BP#1 | .1 BP#2 | .2 WP#1 | .3 WP#2 | .6 Logic Pair#1 | .7 Logic Pair#2 
END_VAR
VAR// IOs 
	SensorBasePos2											: INPUT;
	SensorWorkPos2											: INPUT;
END_VAR

	(* Cylinder	with two inputs for work and base pos each					      	*)
	(* Includes functionblock "INPUT" 												*)
	(********************************************************************************)

(* Write Output *****************************************************)
	IF ToBasePos 	
	THEN
		moveToBasePos();
	ELSIF ToWorkPos AND NOT ToBasePos
	THEN
		moveToWorkPos();
	ELSE
		switchOff();
	END_IF

(* Reedkontakte lesen ***********************************************)
	_readSensors();
	
(* Status *************************************************)
	_writeStatus();
                        	
(* ack Error **********************************************************)
	IF Quit  THEN  reset(); END_IF

(* Timeout  ************************************************)
	_runtimeChk();
	
(*********************************************************************)

METHOD PROTECTED _readSensors : BOOL
VAR_INPUT
END_VAR
(* Call super read sensors first *********************************)
	SUPER^._readSensors();

(* check inputs 2# ************************************************)
	SensorBasePos2(
		Force	:= SensorBasePos.Force ,
		Invert	:= SensorBasePos.Invert,
		PT_ON	:= SensorBasePos.PT_ON,
		PT_OFF	:= SensorBasePos.PT_OFF,
		Q_DIRECT=>,
		Q		=> ,
		Q_RT	=> ,
		Q_FT	=> ,
		IN		=> );


	SensorWorkPos2(
		Force	:= SensorWorkPos.Force,
		Invert	:= SensorWorkPos.Invert,
		PT_ON	:= SensorWorkPos.PT_ON,
		PT_OFF	:= SensorWorkPos.PT_OFF,
		Q_DIRECT=>,
		Q		=> ,
		Q_RT	=> ,
		Q_FT	=> ,
		IN		=> );
		
(* Write status ******************************************)
	InBasePos 									:= SensorBasePos.Q AND SensorBasePos2.Q;
	InWorkPos 									:= SensorWorkPos.Q AND SensorWorkPos2.Q;
	
(* Write error info ***************************************)
	ErrInfo.0									:= TonErrBasePos.Q AND NOT SensorBasePos.Q;
	ErrInfo.1									:= TonErrBasePos.Q AND NOT SensorBasePos2.Q;
	ErrInfo.2									:= TonErrWorkPos.Q AND NOT SensorWorkPos.Q;
	ErrInfo.3									:= TonErrWorkPos.Q AND NOT SensorWorkPos2.Q;

	ErrInfo.6									:= SensorBasePos.Q AND SensorWorkPos.Q;
	ErrInfo.7									:= SensorBasePos2.Q AND SensorWorkPos2.Q;
	
(**************************************************************)
	_readSensors								:= TRUE;
	
(*****************************************************************)
END_METHOD

END_FUNCTION_BLOCK

// ---- POUs/IO/Drives/CoE/AxDriveCoE.TcPOU
{attribute 'no_check'}
//CoE Drive status and diagnosis
//Attention: "SwitchedOn" will be only true if bit 12 "FollowCmdValue" of statusword is used by drive
FUNCTION_BLOCK AxDriveCoE EXTENDS AxDriveBase     
VAR CONSTANT								
END_VAR                  						
VAR_INPUT                           						
	BrakeUnlock												:	BOOL := FALSE;
END_VAR
VAR_IN_OUT
END_VAR
VAR_OUTPUT
	BrakeUnlocked											:	BOOL;
	Status													:	CiA_DS402Statusword;	
	InfoData1										AT %I*	:	UINT;
	InfoData2										AT %I*	:	UINT;
END_VAR                             						
VAR
END_VAR
VAR
(* Cache *********************************************************************)

	// CoE Diagmessage
	StatusTrig												: BYTE;
	MemStatusTrig											: BYTE;
	
(* Timer ********************************************************************************)
  	readDiagDelay											: TON := (PT := T#50MS);
                                  						
(* Trigger ******************************************************************************)


(* Function blocks ****************************************************************************)
	ReadCoEDiagMsg											: EcCoEReadNewestDiagMsg := (Timeout := DEFAULT_ADS_TIMEOUT);	
	CoEWrite												: FB_EcCoeSdoWriteEx := (tTimeout := DEFAULT_ADS_TIMEOUT);	

(* Dummy Speicher **********************************************************)
END_VAR

	(* CoE Drive																		*)
	(************************************************************************************)

(* abort function-call if the reference is invalid *****************************)
IF NOT __ISVALIDREF(rAxis) 
THEN
	Fault													:= TRUE;
	SwitchedOn												:= FALSE;
	Ready													:= FALSE;
	RETURN;         										
END_IF

(* Call super class ****************************************************)
	SUPER^(); 
	
(* Read Statusword ********************************************************)	
	IF rAxis.Status.OpMode.SimulationAxis
	THEN
		IF rAxis.PlcToNc.ControlDWord.0
		THEN
			Status.readStatusword(TO_UINT(eCiA_DS402_STATUS_STATE.OPERATION_ENABLED));
		ELSE
			Status.readStatusword(TO_UINT(eCiA_DS402_STATUS_STATE.SWITCHED_ON));	
		END_IF
	ELSE
		Status.readStatusword(Statusword);
	END_IF			
	
	(* EL72xx DS402 Statusword
		Bit 0 : Ready to switch on
		Bit 1 : Switched on
		Bit 2 : Operation enabled
		Bit 3 : Fault
		Bit 4 : reserved
		Bit 5 : Quick stop (inverse)
		Bit 6 : Switch on disabled
		Bit 7 : Warning
		Bit 8 + 9 : reserved
		Bit 10 : TxPDOToggle (An-/Abwahl über 0x60DA)
		Bit 11 : Internal limit active
		Bit 12 : (drive follows command value)
		Bit 13 - 15 : reserved *)
		
(* DriveStatusBits ***********************************************)
	Fault													:= Status.Fault
																OR rAxis.NcToPlc.StateDWord.28 (* DriveDeviceError *)
																OR rAxis.NcToPlc.StateDWord.30; (* IODataInvalid *)
            												
	Ready 													:= NOT Fault
																AND(Status.ReadyToSwitchOn OR Status.SwitchedOn);

	SwitchedOn												:= Status.SwitchedOn AND NOT Fault;

	
(* manual override brake ********************************************************)
	IF (BrakeUnlock XOR BrakeUnlocked)
		OR CoEWrite.bBusy
	THEN
		BrakeUnlocked										:= BrakeUnlock;
		CoEWrite(
			bExecute	:= NOT CoEWrite.bBusy AND NOT rAxis.NcToPlc.StateDWord.30 AND AdsAddr.port > 0 AND NOT rAxis.Status.OpMode.SimulationAxis,
			sNetId		:= F_CreateAmsNetId(nIds :=AdsAddr.netId),
			nSlaveAddr	:= AdsAddr.port, 
			nIndex		:= 16#8012, 
			nSubIndex	:= 16#1, 
			pSrcBuf		:= ADR(BrakeUnlocked), 
			cbBufLen	:= SIZEOF(BrakeUnlocked));
	END_IF
	
(* Read diagnoses ***********************************************************)
	StatusTrig.0											:= NOT Status.ReadyToSwitchOn;
	StatusTrig.1											:= Status.Fault;
	StatusTrig.2											:= Status.Warning AND NOT Status.Fault;
	
	CASE state OF
	0: // Read subindex of the newest diagnosis message
		
		readDiagDelay(IN := StatusTrig <> MemStatusTrig AND NOT rAxis.Status.OpMode.SimulationAxis AND AdsAddr.port > 0);
	
		IF readDiagDelay.Q
		THEN
			ReadCoEDiagMsg( Execute:= FALSE,  AdsAddr:= AdsAddr);
				
			IF NOT ReadCoEDiagMsg.Busy
			THEN
				MemStatusTrig 								:= StatusTrig; 
				readDiagDelay(IN := FALSE);			
				state 										:= state + 1;
			END_IF
		END_IF
	1: // read newest message
		ReadCoEDiagMsg( Execute:= TRUE,  AdsAddr:= AdsAddr);
		IF NOT ReadCoEDiagMsg.Busy
		THEN
			IF ReadCoEDiagMsg.Error
			THEN
				state										:= 0;
			ELSE	
				state										:= 0;			
			END_IF
			ReadCoEDiagMsg(Execute := FALSE);		
		END_IF
		
	END_CASE
	
(******************************************************************************)

END_FUNCTION_BLOCK

// ---- POUs/IO/Drives/CoE/AxDriveCoE_wEvents.TcPOU
{attribute 'no_check'}
//Drive 
FUNCTION_BLOCK AxDriveCoE_wEvents EXTENDS AxDriveCoE   
VAR_OUTPUT CONSTANT
{attribute 'displaymode':='binary'}  
	OPTION_DISABLE_INT_LIMIT_WARNING						:	BYTE := 2#0000_0001;
{attribute 'displaymode':='binary'}  
	OPTION_DISABLE_REMOTE_CNTR_NOT_ACTIVE					:	BYTE := 2#0000_0010;	
END_VAR                  						
VAR_INPUT                           						
	EnableEvent												:	BOOL := TRUE;
	{attribute 'displaymode':='binary'}  
	Options													:	BYTE := 0;
	ConfirmTrig												:	BOOL := FALSE; (* Reset event *)
	SourceId												:	UDINT := 102200; //CoE Drive default multisource Id + Ax id
	Name													:	STRING(30) := '';
	ErrorLimitPos											:	BOOL := FALSE;
	ErrorLimitNeg											:	BOOL := FALSE;
END_VAR
VAR_IN_OUT
END_VAR
VAR_OUTPUT
	EventStatus												:	DWORD;
	NoOfActiveEvents										:	INT;
END_VAR                             						
VAR

END_VAR
VAR
(* Cache *********************************************************************)
	
(* Timer ********************************************************************************)
                                						
(* Trigger ******************************************************************************)


(* Function blocks ****************************************************************************)
	
	Event													: EventHandlingGrp10;
	EventDiagMessage										: EventHandling;

(* Dummy Speicher **********************************************************)
	i														: INT := 0 ;

END_VAR

	(* CoE Drive with diag and eventlogger implementation								*)
	(************************************************************************************)

(* call super ***********************************************************************)
	SUPER^();

(* trigger events ************************************************)
	_callEvents();

(*****************************************************************)

METHOD _callEvents : BOOL
VAR_INPUT
END_VAR
(* Check if msg activ and init some parameter ***********************)
	IF Event.no[1].Text2 <> Name AND Name <> '' OR Event.no[1].Text2 = '' AND rAxis.NcToPlc.AxisId <> 0
	THEN
		Event.no[1].eClass 									:= TC2_SYSTEM.TCEVENTCLASS_STATEINFO;
		Event.no[3].eClass 									:= TC2_SYSTEM.TCEVENTCLASS_WARNING;
		Event.no[4].eClass 									:= TC2_SYSTEM.TCEVENTCLASS_WARNING;
		Event.no[5].eClass 									:= TC2_SYSTEM.TCEVENTCLASS_STATEINFO;
		Event.no[6].eClass 									:= TC2_SYSTEM.TCEVENTCLASS_STATEINFO;
		Event.no[7].eClass 									:= TC2_SYSTEM.TCEVENTCLASS_STATEINFO;
		
		(* Init axisname *)
		FOR i := Event.MIN_EVENT TO Event.MAX_EVENT DO
		(*	Event.no[i].Text1								:= '';*)
			Event.no[i].Text2								:= SEL(LEN(name)>1,CONCAT('Axis id:',DWORD_TO_STRING(rAxis.NcToPlc.AxisId)),name);			
		END_FOR
		EventDiagMessage.Text2								:= Event.no[1].Text2;
	END_IF

(* workl Event Ctrl *************************************************)
	Event(
		ConfirmTrig 	:= ConfirmTrig,
		Disable			:= rAxis.NcToPlc.AxisId = 0 OR NOT EnableEvent,
		SourceId		:= SourceId + rAxis.NcToPlc.AxisId);
		

(* Event diag message ***************************************************)
	CASE ReadCoEDiagMsg.MsgSeverity OF
	0: // Info message
		EventDiagMessage.eClass 								:= TCEVENTCLASS_MESSAGE;
	1: // warning
		EventDiagMessage.eClass 								:= TCEVENTCLASS_WARNING;
	2: // error message
		EventDiagMessage.eClass 								:= TCEVENTCLASS_ALARM;
	ELSE // unknown type
		EventDiagMessage.eClass 								:= TCEVENTCLASS_NONE;
	END_CASE
				
	EventDiagMessage(
		Flag			:= state = 0 AND ReadCoEDiagMsg.TextId <> 0 AND (Status.Fault OR Status.Warning) AND NOT Event.Disable,
		ConfirmTrig 	:= ConfirmTrig OR NOT EventDiagMessage.Flag AND EventDiagMessage.State <> TCEVENTSTATE_INVALID,
		MsgId			:= ReadCoEDiagMsg.TextId,
		SourceId		:= Event.SourceId);
		
(* Event status ******************************************************)
	NoOfActiveEvents										:= Event.NoOfActiveEvents + SEL(EventDiagMessage.Status.31 , 0, 1);
 	EventStatus												:= Event.Status OR EventDiagMessage.Status;

		
(* Set events at the end to allow set to false in inherited FBs ********************)
	Event.no[1].Flag 										:= NOT Status.ReadyToSwitchOn; 
	Event.no[2].Flag 										:= Status.Fault;
	Event.no[3].Flag 										:= Status.Warning; 				
	Event.no[4].Flag 										:= Status.InternalLimitActive AND NOT Options.0;
	Event.no[5].Flag 										:= Status.SwitchOnDisabled;
//	Event.no[6].Flag 										:= NOT Status.FollowCmdValue AND Status.SwitchedOn AND NOT options.1 AND NOT rAxis.Status.OpMode.SimulationAxis;
	Event.no[7].Flag 										:= BrakeUnlock OR BrakeUnlocked; 	
	Event.no[8].Flag 										:= ErrorLimitPos;
	Event.no[9].Flag 										:= ErrorLimitNeg;
	
(************************************************************************)
	_callEvents												:= TRUE;
(******************************************************************************)
END_METHOD

METHOD PUBLIC confirm : bool
VAR_INPUT
END_VAR
confirm 								:= Event.confirm();
END_METHOD

PROPERTY PUBLIC optDisabledRemoteCntrNotActive : BOOL
GET
optDisabledRemoteCntrNotActive := Options.1;
END_GET
SET
Options.1 := optDisabledRemoteCntrNotActive;
END_SET
END_PROPERTY

PROPERTY PUBLIC optDisableIntLimitWarning : BOOL
GET
optDisableIntLimitWarning := Options.0;
END_GET
SET
Options.0 := optDisableIntLimitWarning;
END_SET
END_PROPERTY

END_FUNCTION_BLOCK

// ---- POUs/IO/Drives/CoE/EL72xx/CiA_DS402StatuswordEx7xxx.TcPOU
FUNCTION_BLOCK CiA_DS402StatuswordEx7xxx EXTENDS CiA_DS402Statusword
VAR_INPUT
END_VAR
VAR_OUTPUT	

	TxPDOToggle				: BOOL; // Bit 10: Following error occured
	FollowCmdValue			: bool;  //Bit 12: Drive follows command (CSP/CSV)
	InputCycleCounter		: BOOL; // Bit 13: 
END_VAR

METHOD PUBLIC readStatusword : BOOL
VAR_INPUT
	Statusword 		:	UINT;
END_VAR
SUPER^.readStatusword(Statusword);

TxPDOToggle													:= Statusword.10;
FollowCmdValue												:= Statusword.12;
InputCycleCounter											:= Statusword.13 ;
	
readStatusword												:= TRUE;
END_METHOD

END_FUNCTION_BLOCK

// ---- POUs/IO/Drives/SoE/AxDriveSoE_Ax5000.TcPOU
{attribute 'no_check'}
//AX5000 SoE drive status and diagnosis FB
FUNCTION_BLOCK AxDriveSoE_Ax5000 extends AxDriveBase (* Lips: TcMc2Drive, TcDrive *)
VAR_INPUT
	ResetTrig												:	BOOL;
	BrakeUnlock												:	BOOL;
	BrakeLock												:	BOOL;					
END_VAR                 									
VAR_IN_OUT              									
END_VAR                 									
VAR_OUTPUT              	                    										
	BrakeStatus												:	BOOL; (* FALSE = OFF / TRUE = ON *)                        								
	RT_StatusChanged										:	BOOL;
{attribute 'displaymode':='binary'}
	MotorsStatusWord										:	WORD; 
	Status													:	ST_AX5000DriveStatus;
	C1D														:	ST_AX5000_C1D;
	DiagMsg 												: 	ST_SoE_String;
	DiagNumber 												: 	UDINT;
	SafetyError										AT %I*	:	BOOL;	(* Ax5805 Drive Safety Error - Bit .7 in Input Safe Data Byte 0 oder 2 *)	
	SercosErrorId											:	UINT;
END_VAR
VAR_OUTPUT CONSTANT
END_VAR
VAR (* EA Internal *)
	(* P-0-0205 - muss ins Zyklische Interface des Reglers unter S-0-0016 (AT) gemappt,
		und dann direkt mit der PLC-Variable verknüpft werden. 
		Oder für das Lesen auf Anforderung die Deklaration auf Lokale Variable ändern 
		und in der Statemaschine für das Status lesen 
		den Auskommentierten Teil mit ins Programm nehmen 
	*)
(*	PwrMgmStatusWord AT %I* : WORD; *)
(*	PwrMgmStatusWord : WORD; *)

END_VAR
VAR

(* Zwischenspeicher *********************************************************************)
	MemDriveStatusword										: 	WORD;
	
	MEM_StatusTrig											:	BYTE;
	StatusTrig												:	BYTE;
	StateReadStatus											:	INT;
	SoEAX5000SetMotorCtrlWordDone							:	BOOL;
	
(* Timer ********************************************************************************)

(* Trigger ******************************************************************************)

(* Bausteine ****************************************************************************)
	SoEAX5000SetMotorCtrlWord 								: FB_SoEAX5000SetMotorCtrlWord_ByDriveRef := (tTimeout := DEFAULT_ADS_TIMEOUT);	(* Bremse manuell lösen *)
	SoEDriveReset											: FB_SoEReset_ByDriveRef := (tTimeout	:= DEFAULT_ADS_TIMEOUT);
	SoERead													: FB_SoERead_ByDriveRef := (tTimeout:= DEFAULT_ADS_TIMEOUT);

(* Dummy Speicher **********************************************************)
	_WORD													: WORD;
	_Dummy													: BOOL;
(****************************************************************************)
END_VAR

	(************************************************************************************)
	(*																					*)
	(*		B E C K H O F F   N E W   A U T O M A T I O N   T E C H N O L O G Y    		*)
	(*																					*)
	(*		Eiserstr.5	D-33415 Verl	Germany	phone:	+49-5246-0	www.Beckhoff.Com	*)
    (*																					*)
    (*		Bausteinbeschreibung	:	AX5000 Drive Ctrl								*)
	(*		TwinCAT-Version			:	3.x or higher 									*)
	(*		Version					:	V3.0 											*)
 	(*		Autor					:	Daniel Schlingmann								*)
	(*		Lib						:	TcMc2Drive.lib / TcDrive.Lib					*)
	(*																					*)
	(************************************************************************************)

(* abort function-call if the reference is invalid *****************************)
IF NOT __ISVALIDREF(rAxis)  THEN
	Fault													:= TRUE;
	Ready													:= FALSE;
	SwitchedOn												:= FALSE;
	RETURN;
END_IF

(* Call super class ****************************************************)
	SUPER^(); 
	
(* DriveStatusword *****************************)
	Status 													:= F_ConvWordToSTAX5000DriveStatus(StatusWord);
	IF rAxis.Status.OpMode.SimulationAxis OR AdsAddr.port = 0
	THEN
		Status.bNotReadyToPowerUp							:= FALSE;	
		Status.bDrvShutdownBitC1D							:= FALSE;
		Status.bReadyForEnable								:= TRUE;
		Status.bEnabled										:= TRUE;	
	END_IF
	(* PowerManagementStatusWord Auswerten *)
	(* Bit 0 = Status UMain ok, ok = True
		Bit 1 = Umain Overvoltage, active = True
		Bit 2 = Umain phase error, error = False
		Bit 3 = Status DcLink ok, ok = True
		Bit 4 = Ext. Umain relay, ready to Switch on = True
		Bit 5 = Status Fan, aktive = True 
		Bit 6 = Status load relay, active = True
		Bit 7 = Status internal chopper, active = True
		Bit 8 = Status external chopper, active = True
		Bit 9 = Status additinal fan, active = True
		Bit 10-15 = reserved *)
	(*
	ReadyForContactor := PowerManagementStatusWord.4;
	*)

(* DriveStatusBits ***********************************************)
	Fault													:= Status.bDrvShutdownBitC1D
																OR rAxis.NcToPlc.StateDWord.28 (* DriveDeviceError *)
																OR rAxis.NcToPlc.StateDWord.30 (* IODataInvalid *)
																OR SafetyError;
            												
	Ready 													:= NOT Fault
																AND(Status.bReadyForEnable OR Status.bEnabled)
																(* AND ReadyForContactor AX 5000 *);

	SwitchedOn												:= Status.bEnabled AND NOT Fault;	
																
(* Init drive ref *************************************************)
	IF AdsAddr.port <> SoEDriveReset.stDriveRef.nSlaveAddr 
	THEN
		SoEDriveReset.stDriveRef.sNetId						:= F_CreateAmsNetId(AdsAddr.netId);	
		SoEDriveReset.stDriveRef.nSlaveAddr					:= AdsAddr.port;	
		SoEDriveReset.stDriveRef.nDriveNo					:= Channel;	
		
		SoEAX5000SetMotorCtrlWord.stDriveRef				:= 	
		SoERead.stDriveRef		 							:= SoEDriveReset.stDriveRef;
	END_IF

(* Reset Drive ****************************************************)
	SoEDriveReset();
	IF SoEDriveReset.bBusy 
	THEN
		; (* Block ist currend working *)
	ELSIF ResetTrig
	THEN
		reset();
	ELSIF SoEDriveReset.bExecute
	THEN
		RefreshStatus();
		SoEDriveReset.bExecute 								:= FALSE;
	END_IF

(* Bremse loesen/setzen  ***********************************************)
	IF (SoEAX5000SetMotorCtrlWord.bForceUnLock XOR BrakeUnlock)
		OR (SoEAX5000SetMotorCtrlWord.bForceLock XOR BrakeLock)
		OR SoEAX5000SetMotorCtrlWord.bBusy 
	THEN
		_Dummy												:= SoEAX5000SetMotorCtrlWord.bBusy;
		SoEAX5000SetMotorCtrlWord(
			stDriveRef	:= ,  //See above
			bExecute	:= NOT SoEAX5000SetMotorCtrlWord.bBusy AND NOT rAxis.Status.OpMode.SimulationAxis, 
			tTimeout	:= , 
			bForceLock	:= BrakeLock , 
			bForceUnlock:= BrakeUnlock , 
			bBusy		=> , 
			bError		=>  , 
			iAdsErrId	=> , 
			iSercosErrId=> );
		SoEAX5000SetMotorCtrlWordDone						:= NOT SoEAX5000SetMotorCtrlWord.bBusy AND _Dummy;
	ELSE 
		SoEAX5000SetMotorCtrlWordDone						:= FALSE;	
	END_IF

(* DriveStatusword auswerten Sercos *****************************)
	RT_StatusChanged 										:= SHR(StatusWord,2) <> MemDriveStatusword OR SoEAX5000SetMotorCtrlWordDone;
	MemDriveStatusword 										:= SHR(StatusWord,2);

(* Start Read Drive status *****************************************************************)
	CASE StateReadStatus OF
	0:
		StatusTrig.0 										:= rAxis.NcToPlc.StateDWord.28;
		StatusTrig.1 										:= rAxis.NcToPlc.StateDWord.30;

		IF NOT rAxis.Status.OpMode.SimulationAxis AND AdsAddr.port > 0
			AND(RT_StatusChanged OR MEM_StatusTrig <> StatusTrig)
		THEN
			refreshStatus();
		ELSE
			;
		END_IF

	(* Read Class 1 Diag *********************************************************)
	10:
		IF NOT SoERead.bBusy
			AND SoERead.bExecute
		THEN
			IF SoERead.bError THEN
				stateReadStatus 							:= 0;
			ELSE                        					
				C1D 										:= F_ConvWordToSTAX5000C1D(_WORD);
				stateReadStatus 							:= stateReadStatus + 1;
			END_IF
		END_IF

		SoERead(
			stDriveRef	:= ,  //See init for drive ref
			nIdn		:= S_0_IDN + 11,
			nElement	:= EC_SOE_ELEMENT_VALUE (* 16#40*),
			pDstBuf		:= ADR(_WORD),
			cbBufLen	:= SIZEOF(_WORD),
			bExecute	:= stateReadStatus = 10,
			tTimeout	:= ,
			bBusy		=> ,
			bError		=> ,
			iAdsErrId	=> ,
			iSercosErrId=> ,
			dwAttribute	=> );

	(* Motor Statusword ***************************************************)
	11:
		IF NOT SoERead.bBusy
			AND SoERead.bExecute
		THEN
			IF SoERead.bError 
			THEN
				stateReadStatus 							:= 0;
			ELSE
				BrakeStatus 								:= MotorsStatusWord.0;
				stateReadStatus 							:= stateReadStatus + 1;
			END_IF
		END_IF

		SoERead(
			stDriveRef	:= ,  //See init for drive ref
			nIdn		:= P_0_IDN + 97, (* Motor Status word *)
			nElement	:= EC_SOE_ELEMENT_VALUE (* 16#40*),
			pDstBuf		:= ADR(MotorsStatusWord),
			cbBufLen	:= SIZEOF(MotorsStatusWord),
			bExecute	:= stateReadStatus = 11,
			tTimeout	:= ,
			bBusy		=> ,
			bError		=> ,
			iAdsErrId	=> ,
			iSercosErrId=> ,
			dwAttribute	=> );


	(* Diag Message *********************************************************)
	12:
		IF NOT SoERead.bBusy
			AND SoERead.bExecute
		THEN
			IF SoERead.bError 
			THEN
				stateReadStatus 							:= 0;
			ELSE
				stateReadStatus 							:= stateReadStatus + 1;
			END_IF
		END_IF

		SoERead(
			stDriveRef	:= ,  //See init for drive ref
			nIdn		:= S_0_IDN + 95,
			nElement	:= EC_SOE_ELEMENT_VALUE (* 16#40*),
			pDstBuf		:= ADR(DiagMsg),
			cbBufLen	:= SIZEOF(DiagMsg),
			bExecute	:= stateReadStatus = 12,
			tTimeout	:= ,
			bBusy		=> ,
			bError		=> ,
			iAdsErrId	=> ,
			iSercosErrId=> ,
			dwAttribute	=> );

	(* Diag Number *********************************************************)
	13:
		IF NOT SoERead.bBusy
			AND SoERead.bExecute
		THEN
			IF SoERead.bError 
			THEN
				stateReadStatus 							:= 0;
			ELSE
				stateReadStatus 							:= stateReadStatus + 1;
			END_IF
		END_IF
		
		SoERead(
			stDriveRef	:= ,  //See init for drive ref
			nIdn		:= S_0_IDN + 390,
			nElement	:= EC_SOE_ELEMENT_VALUE (* 16#40*),
			pDstBuf		:= ADR(DiagNumber),
			cbBufLen	:= SIZEOF(DiagNumber),
			bExecute	:= stateReadStatus = 13,
			tTimeout	:= ,
			bBusy		=> ,
			bError		=> ,
			iAdsErrId	=> ,
			iSercosErrId=> ,
			dwAttribute	=> );

	(* reading status finished ************************************************************)
	ELSE (* Case else *)
		stateReadStatus 									:= 0;
	END_CASE

